(* Logix 5000 project; controller RSL5k_18_Template_noLib Emulate 5570 rev 32.11; software revision 32.02; part 14 of 16 *)
(* tags used below, declared in another part *)
   Inp_SpeedFdbk : REAL;   // Speed Feedbak in Drive Units (typ. 0-32767 = 0 to max freq.)
   Inp_Ready : BOOL;   // 1=Drive is ready to run
   Inp_Running : BOOL;   // 1=Drive is Running (active)
   Inp_CommandDir : BOOL;   // 1=Drive is commanded Forward, 0=Drive is commanded Reverse
   Inp_ActualDir : BOOL;   // 1=Drive is running Forward, 0=Drive is running Reverse
   Inp_FwdPermOK : BOOL;   // 1=Permissives OK, drive can start Forward
   Inp_FwdNBPermOK : BOOL;   // 1=Non-Bypassable Permissives OK, drive can start Forward
   Inp_RevPermOK : BOOL;   // 1=Permissives OK, drive can start Reverse
   Inp_RevNBPermOK : BOOL;   // 1=Non-Bypassable Permissives OK, motor can start Reverse
   Inp_IntlkOK : BOOL;   // 1=Interlocks OK, drive can start/run
   Inp_NBIntlkOK : BOOL;   // 1=Non-Bypassable Interlocks OK, drive can start/run
   Inp_IOFault : BOOL;   // Input Communication Status 0=OK, 1=fail
   Inp_Sim : BOOL;   // 1=Simulate working drive; 0=Start/Stop/ Monitor actual drive
   Inp_OvrdCmd : DINT;   // Override Command: 0=None, 1=Stop, 2=Start Fwd 3=Start Rev
   Cfg_HasRunFdbk : BOOL;   // 1=Drive provides feedback signal on Inp_Running when running
   Cfg_HasSpeedFdbk : BOOL;   // 1=Drive provides speed feedback on Inp_SpeedFdbk
   Cfg_UseSpeedFdbk : BOOL;   // 1=Drive speed determines running state, 0=state determined by drive Active input bit
   Cfg_HasFwdPermObj : BOOL;   // 1=Tells HMI a P_Perm is connected to Inp_FwdPerm
   Cfg_HasRevPermObj : BOOL;   // 1=Tells HMI a P_Perm is connected to Inp_RevPerm
   Cfg_HasIntlkObj : BOOL;   // 1=Tells HMI a P_Intlk is connected to Inp_Intlk
   Cfg_HasResInhObj : BOOL;   // 1=Tells HMI a P_ResInh Restart Inhibit is connected
   Cfg_HasRunTimeObj : BOOL;   // 1=Tells HMI a P_RunTime is connected
   Cfg_SetTrack : BOOL;   // 1=Settings track for unselected sources, 0=no tracking
   Cfg_ShedOnFailToStart : BOOL;   // 1=Stop Motor and Alarm on Fail to Start; 0=Alarm only on Fail to Start
   Cfg_ShedOnIOFault : BOOL;   // 1=Stop Motor and Alarm on I/O Fault; 0=Alarm only on I/O Fault
   Cfg_DecPlcs : DINT;   // Number of decimal places for speed ref/fdbk display (0..6)
   Cfg_InpDLDecPlcs : DINT;   // Number of decimal places for Input Datalink display (0..6)
   Cfg_OutDLDecPlcs : DINT;   // Number of decimal places for Output Datalink display (0..6)
   Cfg_HasDriveFaultAlm : ALIAS FOR DriveFault.Cfg_Exists;   // 1=Drive Fault alarm exists and will be checked
   Cfg_DriveFaultResetReqd : ALIAS FOR DriveFault.Cfg_ResetReqd;   // 1=Reset required to clear Drive Fault Alarm
   Cfg_FailToStartAckReqd : ALIAS FOR FailToStart.Cfg_AckReqd;   // 1=Acknowledge required for Fail to Start Alarm
   Cfg_FailToStopAckReqd : ALIAS FOR FailToStop.Cfg_AckReqd;   // 1=Acknowledge required for Fail to Stop Alarm
   Cfg_IntlkTripAckReqd : ALIAS FOR IntlkTrip.Cfg_AckReqd;   // 1=Acknowledge required for Interlock Trip Alarm
   Cfg_DriveFaultAckReqd : ALIAS FOR DriveFault.Cfg_AckReqd;   // 1=Acknowledge required for Drive Fault Alarm
   Cfg_IOFaultAckReqd : ALIAS FOR IOFault.Cfg_AckReqd;   // 1=Acknowledge required for I/O Fault Alarm
   Cfg_FailToStartSeverity : ALIAS FOR FailToStart.Cfg_Severity;   // Fail To Start Alarm Severity: 1..250=Low, 251..500=Medium, 501..750=High, 751..1000=Urgent
   Cfg_FailToStopSeverity : ALIAS FOR FailToStop.Cfg_Severity;   // Fail To Stop Alarm Severity: 1..250=Low, 251..500=Medium, 501..750=High, 751..1000=Urgent
   Cfg_IntlkTripSeverity : ALIAS FOR IntlkTrip.Cfg_Severity;   // Interlock Trip Alarm Severity: 1..250=Low, 251..500=Medium, 501..750=High, 751..1000=Urgent
   Cfg_DriveFaultSeverity : ALIAS FOR DriveFault.Cfg_Severity;   // Drive Fault Alarm Severity: 1..250=Low, 251..500=Medium, 501..750=High, 751..1000=Urgent
   Cfg_IOFaultSeverity : ALIAS FOR IOFault.Cfg_Severity;   // I/O Fault Alarm Severity: 1..250=Low, 251..500=Medium, 501..750=High, 751..1000=Urgent
   Cfg_MaxSpdRef : REAL;   // Maximum Speed Reference in EU (for limiting)
   Cfg_SpeedRefRawMax : REAL;   // Speed Reference Maximum in Drive (raw) Units (for scaling)
   Cfg_SpeedRefEUMax : REAL;   // Speed Reference Maximum in Engineering Units (for scaling)
   Cfg_SpeedFdbkRawMax : REAL;   // Speed Feedback Maximum in Drive (raw) Units (for scaling)
   Cfg_SpeedFdbkEUMax : REAL;   // Speed Feedback Maximum in Engineering Units (for scaling)
   Cfg_InpDatalinkRawMax : REAL;   // Input Datalink Maximum in Drive (raw) Units (for scaling)
   Cfg_InpDatalinkEUMax : REAL;   // Input Datalink Maximum in Engineering Units (for scaling)
   Cfg_OutDatalinkMax : REAL;   // Maximum Output Datalink in EU (for limiting)
   Cfg_OutDatalinkRawMax : REAL;   // Output Datalink Maximum in Drive (raw) Units (for scaling)
   Cfg_OutDatalinkEUMax : REAL;   // Output Datalink Maximum in Engineering Units (for scaling)
   Cfg_SimRampT : REAL;   // Time to ramp speed fdbk when in Simulation (sec)
   Cfg_FailToStartT : REAL;   // Time after Start to get Run Feedback before Fault (sec)
   Cfg_FailToStopT : REAL;   // Time after Stop to drop Run Feedback before Fault (sec)
   Cfg_ResetPulseT : REAL;   // Time to pulse Out_Reset to clear drive fault
   Cfg_OperKeep : SINT;   // Oper keeps control in Prog / Ext: .0=Reference, .1=Start/Stop/Fwd/ Rev, .3=OutDatalink
   Cfg_ProgKeep : SINT;   // Prog keeps control in Oper / Ext: .0=Reference, .1=Start/Stop/Fwd/ Rev, .3=OutDatalink
   Cfg_ExtKeep : SINT;   // Ext keeps control in Prog / Oper: .0=Reference, .1=Start/Stop/Fwd/ Rev, .3=OutDatalink
   PSet_SpeedRef : REAL;   // Program Setting of Speed Reference (EU)
   PSet_Owner : DINT;   // Program Owner Request ID (non-zero) or Release (zero)
   XSet_SpeedRef : REAL;   // External Setting of Speed Reference (EU)
   PCmd_StartFwd : BOOL;   // Program Command to Start Drive Forward
   PCmd_StartRev : BOOL;   // Program Command to Start Drive Reverse
   PCmd_Stop : BOOL;   // Program Command to Stop Drive
   PCmd_Reset : BOOL;   // Program Command to Reset drive fault and all Alarms requiring Reset
   XCmd_StartFwd : BOOL;   // External Command to Start Drive Forward
   XCmd_StartRev : BOOL;   // External Command to Start Drive Reverse
   XCmd_Stop : BOOL;   // External Command to Stop Drive
   XCmd_JogFwd : BOOL;   // External Command to Jog Drive Forward
   XCmd_JogRev : BOOL;   // External Command to Jog Drive Reverse
   XCmd_Reset : BOOL;   // Ext Cmd to clear shed latches and cleared alarms
   Out_SpeedRef : REAL;   // Drive Speed Reference in Drive Units (typ. 0-32767 = 0 to max freq.)
   Out_Datalink : REAL;   // Auxiliary Signal (datalink) Output in Drive (raw) Units
   Out_Run : BOOL;   // 1=Start/Run Drive, 0=Stop Drive (for held starter type)
   Out_Stop : BOOL;   // 1=Stop Drive, 0=drive left in current state
   Out_Start : BOOL;   // 1=Start Drive, 0=drive left in current state
   Out_Jog : BOOL;   // 1=Jog drive at Jog Speed, -->0=stop jogging
   Out_ClearFault : BOOL;   // 1=Attempt to clear Drive Fault
   Out_Fwd : BOOL;   // 1=Set drive direction to Forward
   Out_Rev : BOOL;   // 1=Set drive direction to Reverse
   Out_Horn : BOOL;   // 1=Sound audible prior to commanded motor start
   Val_SpeedRef : REAL;   // Speed Reference (target) to drive
   Val_SpeedFdbk : REAL;   // Speed Feedback (actual) from drive
   Val_SpeedRefEUMax : REAL;   // Maximum of Speed Reference = MAX (Cfg_SpeedFdbkEUMin, Cfg_SpeedFdbkEUMax)
   Val_SpeedFdbkEUMax : REAL;   // Maximum of Speed Feedback = MAX (Cfg_SpeedFdbkEUMin, Cfg_SpeedFdbkEUMax)
   SrcQ_IO : DINT;   // Source and Quality of primary I/O (enumeration)
   SrcQ : DINT;   // Source and Quality of primary Val/Sts (enumeration)
   Val_Cmd : DINT;   // Device Command 0=None, 1=Stop, 2=StartFwd 3=StartRev 4=JogFwd 5=JogRev
   Val_Fdbk : DINT;   // Device Feedback 0=Stopped, 1=Running Fwd 2=Running Rev 3=Accelerating 4=Decelerating
   Val_Sts : DINT;   // Device Sts: 0=? 1=Stopped 2=RunFwd 3=RunRev 4=RunSlow 5=StartFwd 6=StartRev 7=StartSlow 8=JogFwd 9=JogRev 10=Stopping
   Val_Fault : DINT;   // Device Fault Status 0=None, 16=Fail to Start, 17 = Fail to Stop, 18=Drive Fault, 32=I/O Fault, 34=Config Error
   Val_NotifyAll : DINT;   // Highest Alarm prio and ack status this object + channel (enum)
   Val_UnackAlmC : DINT;   // Count of Unacknowledged Alarms
   Val_Owner : DINT;   // Current Object Owner ID (0=not owned)
   Sts_Stopped : BOOL;   // 1=Drive requested to stop and is confirmed stopped
   Sts_StartingFwd : BOOL;   // 1=Drive requested to run forward and awaiting run feedback
   Sts_StartingRev : BOOL;   // 1=Drive requested to run reverse and awaiting run feedback
   Sts_RunningFwd : BOOL;   // 1=Drive requested to run and is confirmed running forward
   Sts_RunningRev : BOOL;   // 1=Drive requested to run and is confirmed running reverse
   Sts_StoppingFwd : BOOL;   // 1=Drive running forward requested to stop and awaiting stopped feedback
   Sts_StoppingRev : BOOL;   // 1=Drive running reverse requested to stop and awaiting stopped feedback
   Sts_JoggingFwd : BOOL;   // 1=Drive requested to Jog Forward
   Sts_JoggingRev : BOOL;   // 1=Drive requested to Jog Reverse
   Sts_Horn : BOOL;   // 1=Motor Horn Active
   Sts_CommandDir : BOOL;   // 1=Drive commanded to Forward, 0=Reverse
   Sts_ActualDir : BOOL;   // 1=Drive Actual direction is Forward, 0=Reverse
   Sts_Available : BOOL;   // 1=Drive available for control by automation (Prog)
   Nrdy_CfgErr : BOOL;   // 1=Device Not Ready: Configuration Error
   Nrdy_Fail : BOOL;   // 1=Device Not Ready: Device Failure (Shed Requires Reset)
   Nrdy_IOFault : BOOL;   // 1=Device Not Ready: I/O Fault (Shed Requires Reset)
   Nrdy_PrioStop : BOOL;   // 1=Device Not Ready: Oper/Ext Priority Stop Requires Reset
   Nrdy_Trip : BOOL;   // 1=Device not Ready: Deivce Tripped (Drive Fault)
   Sts_Err : BOOL;   // 1=Error in Config: see detail bits for reason
   Err_Alarm : BOOL;   // 1=Error in Config: Alarm Min On Time, Shelf Time, Severity
   Err_FdbkRaw : BOOL;   // 1=Erron in Config: Speed Fdbk Raw Min = Max
   Err_FdbkEU : BOOL;   // 1=Error in Config: Speed Fdbk EU Min = Max
   Sts_Prog : ALIAS FOR CmdSrc.Sts_Prog;
   Sts_Oper : ALIAS FOR CmdSrc.Sts_Oper;
   Sts_Normal : ALIAS FOR CmdSrc.Sts_Normal;
   Sts_ExtReqInh : ALIAS FOR CmdSrc.Sts_ExtReqInh;
   Sts_RdyReset : ALIAS FOR ORdy_Reset;   // 1=A latched alarm or shed condition is ready to be reset
   Sts_RdyAck : BOOL;   // 1=An alarm is ready to be acknowledged
   Ack_FailToStart : ALIAS FOR FailToStart.Ack;   // 1=Fail to Start Alarm has been acknowledged
   Sts_FailToStop : ALIAS FOR FailToStop.Inp;   // 1=Drive Failed to Stop
   Ack_FailToStop : ALIAS FOR FailToStop.Ack;   // 1=Fail to Stop Alarm has been acknowledged
   Ack_IntlkTrip : ALIAS FOR IntlkTrip.Ack;   // 1=Interlock Trip Alarm has been acknowledged
   Sts_DriveFault : ALIAS FOR DriveFault.Inp;   // 1=Drive Fault (see drive display or manual)
   Ack_DriveFault : ALIAS FOR DriveFault.Ack;   // 1=Drive Fault Alarm has been acknowledged
   Sts_IOFault : ALIAS FOR IOFault.Inp;   // I/O Comm Fault Status (0=OK, 1=Bad)
   Ack_IOFault : ALIAS FOR IOFault.Ack;   // 1=I/O Fault Alarm has been acknowledged
   P_VSD : BOOL;   // Unique Parameter Name for auto - discovery
   IOFault : P_Alarm;   // I/O Fault Alarm
   IntlkTrip : P_Alarm;   // Interlock Trip Alarm
   FailToStop : P_Alarm;   // Drive Failed to Stop Alarm
   FailToStart : P_Alarm;   // Drive Failed to Start Alarm
   Wrk_Run : BOOL;   // 1=Drive should be "running", 0=should be "stopped"
   Wrk_Notify : DINT;   // Buffer for building Val_Notify
   DriveFault : P_Alarm;   // Drive Faulted Alarm
   Wrk_Jog : BOOL;   // 1=Jog Drive, 0=Drive not jogging
   Wrk_Sts : DINT;   // Buffer for building Val_Sts
   Wrk_Fault : DINT;   // Buffer for building Val_Fault
   Wrk_SrcQ : DINT;   // Register for building Source / Quality enumeration
   Val_Notify : DINT;   // Current Alarm Level and Acknowledgement (enumeration)
   Wrk_UnackAlmC : DINT;   // Buffer for building Val_UnackAlmC
   OCmd_ResetAckAll : BOOL;   // Oper Cmd to reset shed latches and cleared alarms, plus Acknowledge alarms
   OCmd_Reset : BOOL;   // Oper Cmd to clear shed latches and cleared alarms
   OCmd_JogRev : BOOL;   // Operator Command to Jog Drive Reverse (not cleared by instruction!)
   OCmd_JogFwd : BOOL;   // Operator Command to Jog Drive Forward (not cleared by instruction!)
   OCmd_Stop : BOOL;   // Operator Command to Stop Drive
   OCmd_StartRev : BOOL;   // Operator Command to Start Drive Reverse
   OCmd_StartFwd : BOOL;   // Operator Command to Start Drive Forward
   MCmd_Check : BOOL;   // Maintenance Command to Check (not bypass) all Interlocks and Permissives
   MCmd_Bypass : BOOL;   // Maintenance Command to Bypass all Bypassable Interlocks and Permissives
   ORdy_ResetAckAll : BOOL;   // 1=Ready for OCmd_ResetAckAll (enables HMI button)
   ORdy_Reset : BOOL;   // 1=Ready for OCmd_Reset (enables HMI button)
   ORdy_JogRev : BOOL;   // 1=Ready for OCmd_JogRev (enabled HMI button)
   ORdy_JogFwd : BOOL;   // 1=Ready for OCmd_JogFwd (enables HMI button)
   ORdy_Stop : BOOL;   // 1=Ready for OCmd_Stop (enables HMI button)
   ORdy_StartRev : BOOL;   // 1=Ready for OCmd_StartRev (enables HMI button)
   ORdy_StartFwd : BOOL;   // 1=Ready for OCmd_StartFwd (enables HMI button)
   ORdy_SpeedRef : BOOL;   // 1=Ready for OSet_SpeedRef (enables data entry field)
   MRdy_Check : BOOL;   // 1=Ready for MCmd_Check (enables HMI button)
   MRdy_Bypass : BOOL;   // 1=Ready for MCmd_Bypass (enables HMI button)
(* P_VSD, continued *)

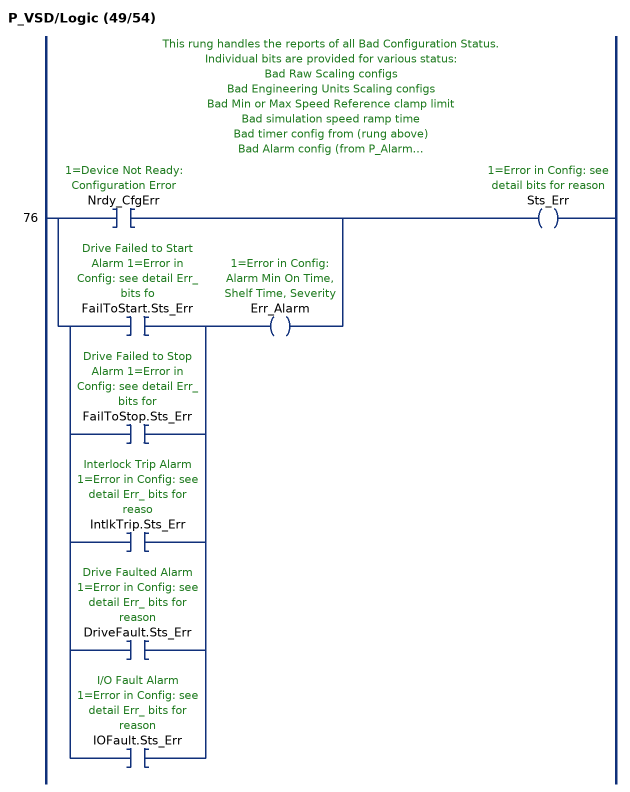
   // This rung handles the reports of all Bad Configuration Status.
   // Individual bits are provided for various status:
   // Bad Raw Scaling configs
   // Bad Engineering Units Scaling configs
   // Bad Min or Max Speed Reference clamp limit
   // Bad simulation speed ramp time
   // Bad timer config from (rung above)
   // Bad Alarm config (from P_Alarm)
   // Bad Cfg_OperKeep / Cfg_ProgKeep config
   // Then a summary Bad Config status is provided, simply an OR of the individual bits.
   // #####  V4.00.00  2018-07-13:  Modified to allow the special case where min and max clamping  #####
   // #####  limits (speed or output datalink) can be EQUAL (clamp at a specific value).  #####
   // #####  Changed delay / time configuration items to REAL seconds.  #####
   76: [XIC(Nrdy_CfgErr) ,[XIC(FailToStart.Sts_Err) ,XIC(FailToStop.Sts_Err) ,XIC(IntlkTrip.Sts_Err) ,XIC(DriveFault.Sts_Err) ,XIC(IOFault.Sts_Err) ] OTE(Err_Alarm) ]OTE(Sts_Err);
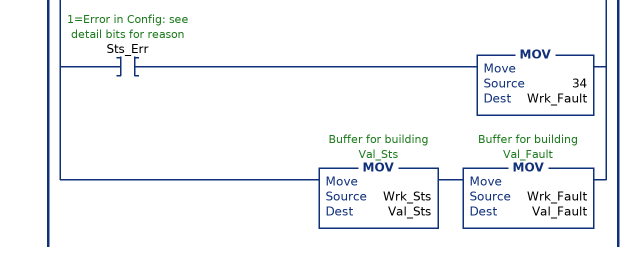
   // Val_Sts is the current device status, as determined by this AOI,
   // based on its knowledge of commands executed and feedback.
   // (This is the status that should be monitored by, for example, FT Historian.)
   // 0 = Powerup / Unknown (in Hand but having no feedback, for example)
   // 0 = Powerup / Unknown
   // 1 = Stopped
   // 2 = Running Forward
   // 3 = Running Reverse
   // 4 = Running Slow
   // 5 = Starting Forward
   // 6 = Starting Reverse
   // 7 = Starting Slow
   // 8 = Jogging Forward
   // 9 = Jogging Reverse
   // 10 = Stopping
   // 14 = Horn
   // Val_Fault is the current device fault status, as determined by this AOI,
   // based on its knowledge of commands executed and feedback.
   // (This is the fault status that should be monitored by, for example, FT Historian.)
   // 0 = None
   // 16 = Fail to Start
   // 17 = Fail to Stop
   // 18 = Drive Fault
   // 32 = I/O Fault (from Input)
   // 34 = Configuration Error
   // #####  V4.00.00 2018-07-13:  Changed Start / Stop / Jog / Fwd / Rev to StartFwd / StartRev / Stop / JogFwd / JogRev  #####
   // #####  Disable/Enable replaced by P_CmdSrc Out of Service (OoS).  #####
   // #####  V4.10.00  2019-03-25:  Added Horn Status.  #####
   77: [CLR(Wrk_Sts) CLR(Wrk_Fault) ,XIC(Sts_Stopped) MOV(1,Wrk_Sts) ,XIC(Sts_RunningFwd) MOV(2,Wrk_Sts) ,XIC(Sts_RunningRev) MOV(3,Wrk_Sts) ,XIC(Sts_StartingFwd) MOV(5,Wrk_Sts) ,XIC(Sts_StartingRev) MOV(6,Wrk_Sts) ,XIC(Sts_JoggingFwd) MOV(8,Wrk_Sts) ,XIC(Sts_JoggingRev) MOV(9,Wrk_Sts) ,[XIC(Sts_StoppingFwd) ,XIC(Sts_StoppingRev) ] MOV(10,Wrk_Sts) ,XIC(Sts_Horn) MOV(14,Wrk_Sts) ,XIC(Nrdy_Fail) MOV(16,Wrk_Fault) ,XIC(Sts_FailToStop) MOV(17,Wrk_Fault) ,XIC(Sts_DriveFault) MOV(18,Wrk_Fault) ,[XIC(Sts_IOFault) ,XIC(Nrdy_IOFault) ] MOV(32,Wrk_Fault) ,XIC(Sts_Err) MOV(34,Wrk_Fault) ,MOV(Wrk_Sts,Val_Sts) MOV(Wrk_Fault,Val_Fault) ];
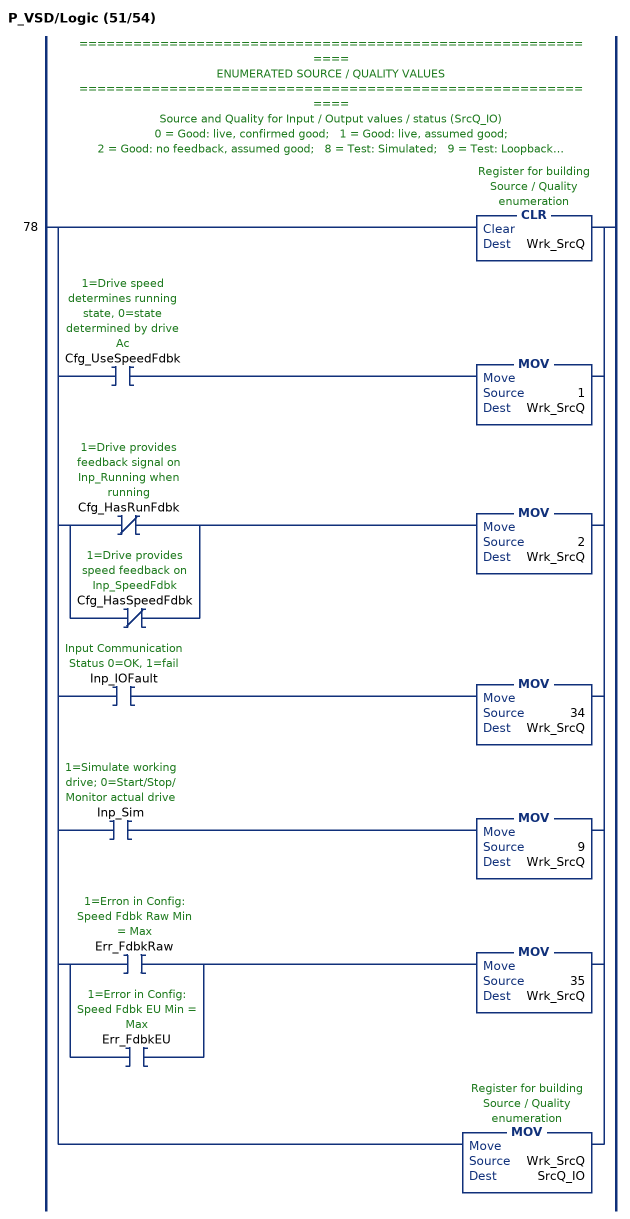
   // ============================================================
   // ENUMERATED SOURCE / QUALITY VALUES
   // ============================================================
   // Source and Quality for Input / Output values / status (SrcQ_IO)
   // 0 = Good: live, confirmed good;   1 = Good: live, assumed good;
   // 2 = Good: no feedback, assumed good;   8 = Test: Simulated;   9 = Test: Loopback;
   // 10 = Test: Manually Entered;   16 = Uncertain: Live, off-spec;
   // 17 = Uncertain, Substituted at Device / Bus;   18 = Uncertain, Substituted at AOI;
   // 19 = Uncertain, using last known good;    20 = Uncertain, using replacement value;
   // 32 = Bad, Signal Failure;   33 = Bad, Channel Fault;
   // 34 = Bad, Module / Comms Fault;   35 = Bad, Invalid Configuration
   78: [CLR(Wrk_SrcQ) ,XIC(Cfg_UseSpeedFdbk) MOV(1,Wrk_SrcQ) ,[XIO(Cfg_HasRunFdbk) ,XIO(Cfg_HasSpeedFdbk) ] MOV(2,Wrk_SrcQ) ,XIC(Inp_IOFault) MOV(34,Wrk_SrcQ) ,XIC(Inp_Sim) MOV(9,Wrk_SrcQ) ,[XIC(Err_FdbkRaw) ,XIC(Err_FdbkEU) ] MOV(35,Wrk_SrcQ) ,MOV(Wrk_SrcQ,SrcQ_IO) ];
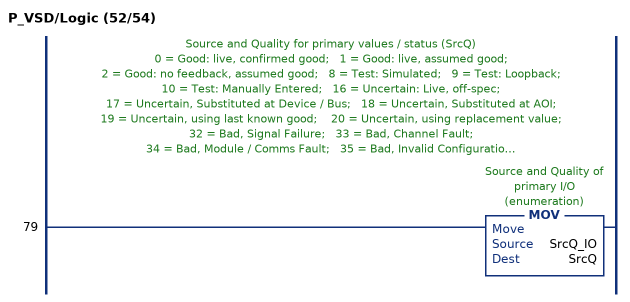
   // Source and Quality for primary values / status (SrcQ)
   // 0 = Good: live, confirmed good;   1 = Good: live, assumed good;
   // 2 = Good: no feedback, assumed good;   8 = Test: Simulated;   9 = Test: Loopback;
   // 10 = Test: Manually Entered;   16 = Uncertain: Live, off-spec;
   // 17 = Uncertain, Substituted at Device / Bus;   18 = Uncertain, Substituted at AOI;
   // 19 = Uncertain, using last known good;    20 = Uncertain, using replacement value;
   // 32 = Bad, Signal Failure;   33 = Bad, Channel Fault;
   // 34 = Bad, Module / Comms Fault;   35 = Bad, Invalid Configuration
   // If the drive is using run feedback (for state) and has speed feedback, all is live and good.
   // If the drive is using speed feedback to determine run state, state is assumed good.
   // If the drive does not have speed feedback, speed is no-feedback assumed good.
   79: MOV(SrcQ_IO,SrcQ);
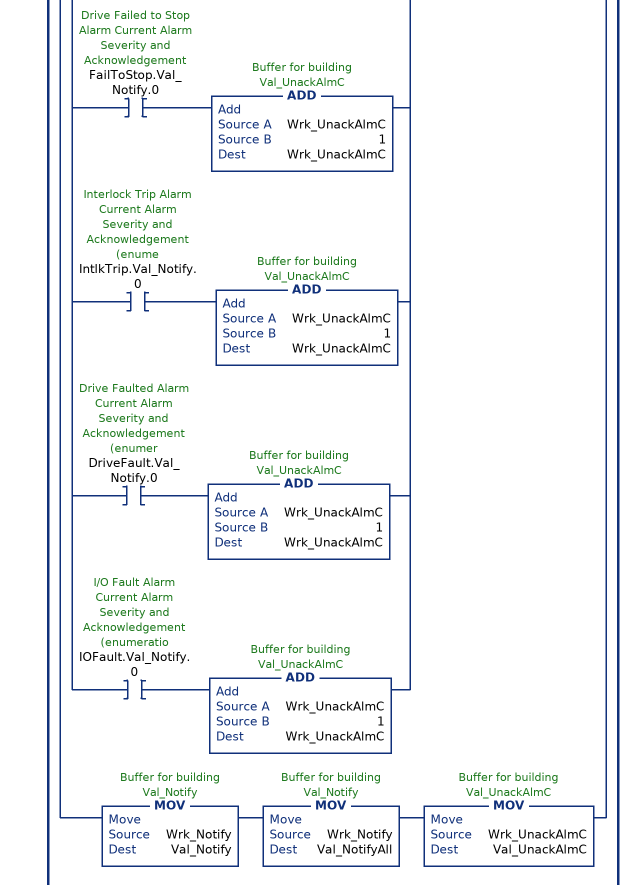
   // ============================================================
   // NOTIFICATION VALUE
   // ============================================================
   // Indicate the current alarm notification level as the max of any of the alarms,
   // and set the low-order bit for reset or ack required:
   // 0 = Not in alarm, acknowledged
   // 1 = Not in alarm, unacknowledged or reset required
   // 2 = Low severity alarm, acknowledged
   // 3 = Low severity alarm, unacknowledged
   // 4 = Medium severity alarm, acknowledged
   // 5 = Medium severity alarm, unacknowledged
   // 6 = High severity alarm, acknowledged
   // 7 = High severity alarm, unacknowledged
   // 8 = Urgent severity alarm, acknowledged
   // 9 = Urgent severity alarm, unacknowledged
   // #####  V4.00.00  2018-07-13:  Added Val_NotifyAll and Val_UnackAlmC to roll up alarm  #####
   // #####  priority / ack status and unack. alarm count.  #####
   80: [CLR(Wrk_Notify) CLR(Wrk_UnackAlmC) ,GRT(FailToStart.Val_Notify,Wrk_Notify) MOV(FailToStart.Val_Notify,Wrk_Notify) ,GRT(FailToStop.Val_Notify,Wrk_Notify) MOV(FailToStop.Val_Notify,Wrk_Notify) ,GRT(IntlkTrip.Val_Notify,Wrk_Notify) MOV(IntlkTrip.Val_Notify,Wrk_Notify) ,GRT(DriveFault.Val_Notify,Wrk_Notify) MOV(DriveFault.Val_Notify,Wrk_Notify) ,GRT(IOFault.Val_Notify,Wrk_Notify) MOV(IOFault.Val_Notify,Wrk_Notify) ,[XIC(FailToStart.Val_Notify.0) ADD(Wrk_UnackAlmC,1,Wrk_UnackAlmC) ,XIC(FailToStop.Val_Notify.0) ADD(Wrk_UnackAlmC,1,Wrk_UnackAlmC) ,XIC(IntlkTrip.Val_Notify.0) ADD(Wrk_UnackAlmC,1,Wrk_UnackAlmC) ,XIC(DriveFault.Val_Notify.0) ADD(Wrk_UnackAlmC,1,Wrk_UnackAlmC) ,XIC(IOFault.Val_Notify.0) ADD(Wrk_UnackAlmC,1,Wrk_UnackAlmC) ] OTE(Wrk_Notify.0) ,MOV(Wrk_Notify,Val_Notify) MOV(Wrk_Notify,Val_NotifyAll) MOV(Wrk_UnackAlmC,Val_UnackAlmC) ];
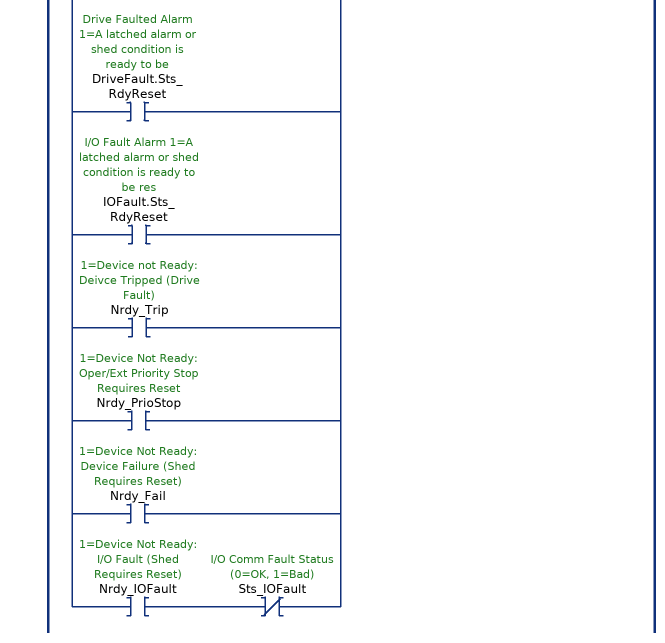
   // This rung identifies:
   // * if a latched Shed condition requires a reset in order to run the motor;
   // * if that reset or any alarm reset or other reset is required; and
   // * if any reset or acknowledge from the operator is required.
   // #####  V4.00.00  2018-07-13:  Aligned ready bit naming with command bit names.  #####
   // #####  All OCmds/MCmds and ORdys/MRdys are now Local Tags.  #####
   // #####  Added Sts_RdyAck and Sts_ResetReqd for use by external objects.  #####
   81: [[XIC(FailToStart.Sts_RdyAck) ,XIC(FailToStop.Sts_RdyAck) ,XIC(IntlkTrip.Sts_RdyAck) ,XIC(IOFault.Sts_RdyAck) ,XIC(DriveFault.Sts_RdyAck) ] OTE(Sts_RdyAck) ,[XIC(FailToStart.Sts_RdyReset) ,XIC(FailToStop.Sts_RdyReset) ,XIC(IntlkTrip.Sts_RdyReset) ,XIC(DriveFault.Sts_RdyReset) ,XIC(IOFault.Sts_RdyReset) ,XIC(Nrdy_Trip) ,XIC(Nrdy_PrioStop) ,XIC(Nrdy_Fail) ,XIC(Nrdy_IOFault) XIO(Sts_IOFault) ] OTE(ORdy_Reset) ]OTE(ORdy_ResetAckAll);
END_ROUTINE

ROUTINE Prescan   (* ladder *)
// Clear Ownership, set drive to STOP, clear "lurking" Commands
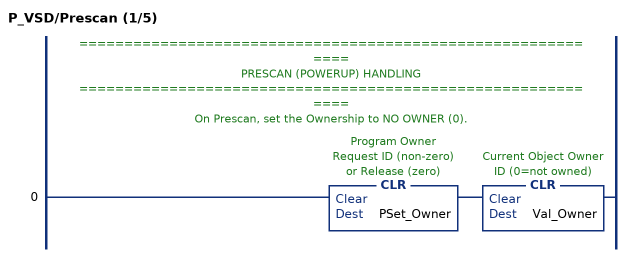
   // ============================================================
   // PRESCAN (POWERUP) HANDLING
   // ============================================================
   // On Prescan, set the Ownership to NO OWNER (0).
   0: CLR(PSet_Owner)CLR(Val_Owner);
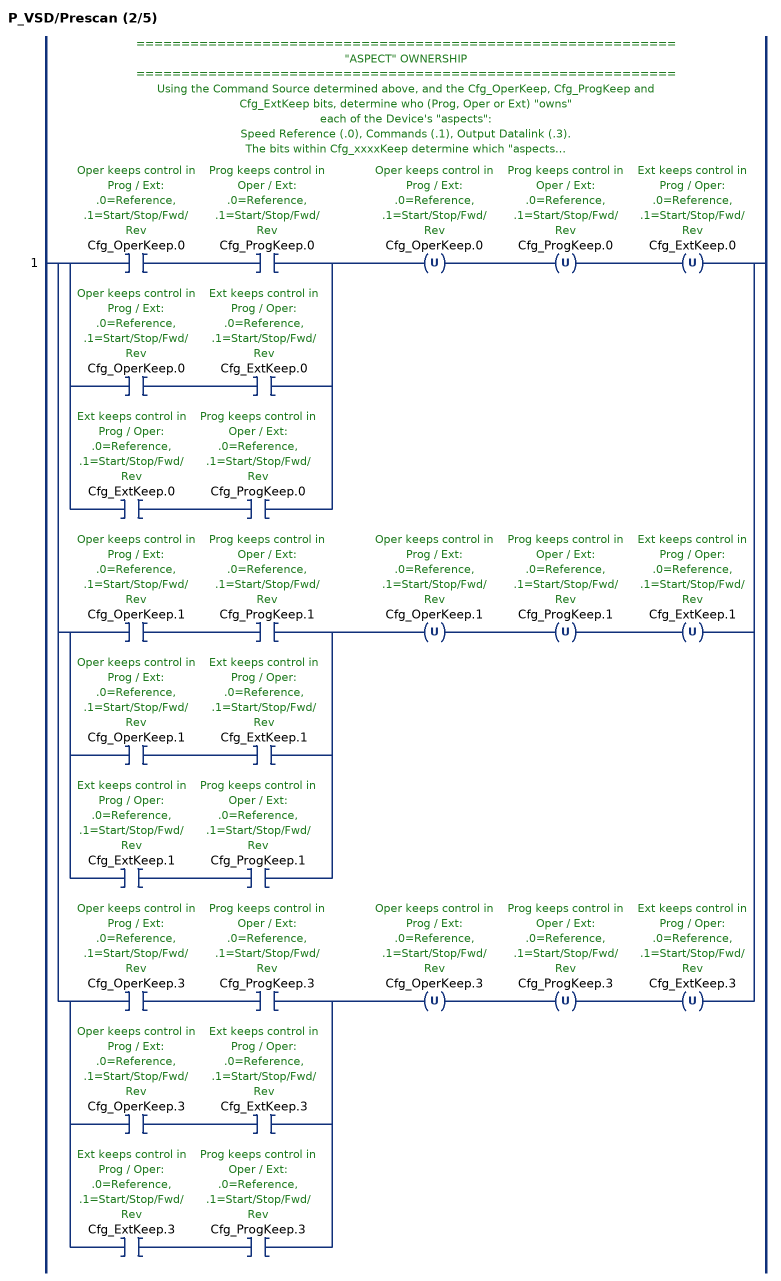
   // ============================================================
   // "ASPECT" OWNERSHIP
   // ============================================================
   // Using the Command Source determined above, and the Cfg_OperKeep, Cfg_ProgKeep and
   // Cfg_ExtKeep bits, determine who (Prog, Oper or Ext) "owns"
   // each of the Device's "aspects":
   // Speed Reference (.0), Commands (.1), Output Datalink (.3).
   // The bits within Cfg_xxxxKeep determine which "aspects"
   // (sub-functions of this AOI) are retained by the Oper, Prog or Ext
   // when one of the other command sources is selected.
   // All aspects (functions) may be "kept" (basically locking the command source
   // slection, rendering it moot --  you get to explain how it works to your operators!!!),
   // but it is NOT allowed to have any given function retained by more than one
   // source.  This rung ensures that no function is "kept" by more than one source.
   // ON PRESCAN:  If any two of Oper Keep, Prog Keep and Ext Keep get set on download or during
   // controller PROG mode, they are ALL CLEARED on powerup!!!
   1: [[XIC(Cfg_OperKeep.0) XIC(Cfg_ProgKeep.0) ,XIC(Cfg_OperKeep.0) XIC(Cfg_ExtKeep.0) ,XIC(Cfg_ExtKeep.0) XIC(Cfg_ProgKeep.0) ] OTU(Cfg_OperKeep.0) OTU(Cfg_ProgKeep.0) OTU(Cfg_ExtKeep.0) ,[XIC(Cfg_OperKeep.1) XIC(Cfg_ProgKeep.1) ,XIC(Cfg_OperKeep.1) XIC(Cfg_ExtKeep.1) ,XIC(Cfg_ExtKeep.1) XIC(Cfg_ProgKeep.1) ] OTU(Cfg_OperKeep.1) OTU(Cfg_ProgKeep.1) OTU(Cfg_ExtKeep.1) ,[XIC(Cfg_OperKeep.3) XIC(Cfg_ProgKeep.3) ,XIC(Cfg_OperKeep.3) XIC(Cfg_ExtKeep.3) ,XIC(Cfg_ExtKeep.3) XIC(Cfg_ProgKeep.3) ] OTU(Cfg_OperKeep.3) OTU(Cfg_ProgKeep.3) OTU(Cfg_ExtKeep.3) ];
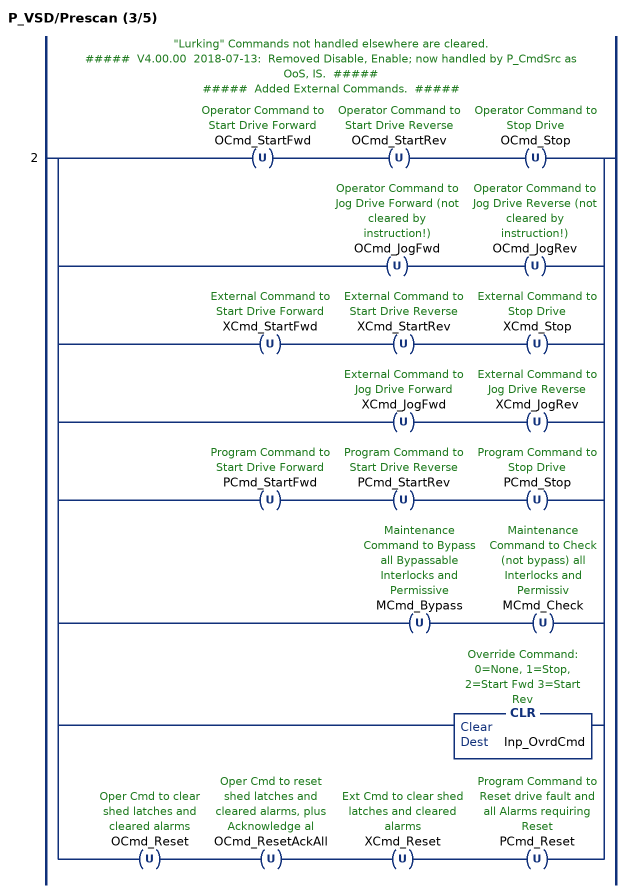
   // "Lurking" Commands not handled elsewhere are cleared.
   // #####  V4.00.00  2018-07-13:  Removed Disable, Enable; now handled by P_CmdSrc as OoS, IS.  #####
   // #####  Added External Commands.  #####
   2: [OTU(OCmd_StartFwd) OTU(OCmd_StartRev) OTU(OCmd_Stop) ,OTU(OCmd_JogFwd) OTU(OCmd_JogRev) ,OTU(XCmd_StartFwd) OTU(XCmd_StartRev) OTU(XCmd_Stop) ,OTU(XCmd_JogFwd) OTU(XCmd_JogRev) ,OTU(PCmd_StartFwd) OTU(PCmd_StartRev) OTU(PCmd_Stop) ,OTU(MCmd_Bypass) OTU(MCmd_Check) ,CLR(Inp_OvrdCmd) ,OTU(OCmd_Reset) OTU(OCmd_ResetAckAll) OTU(XCmd_Reset) OTU(PCmd_Reset) ];
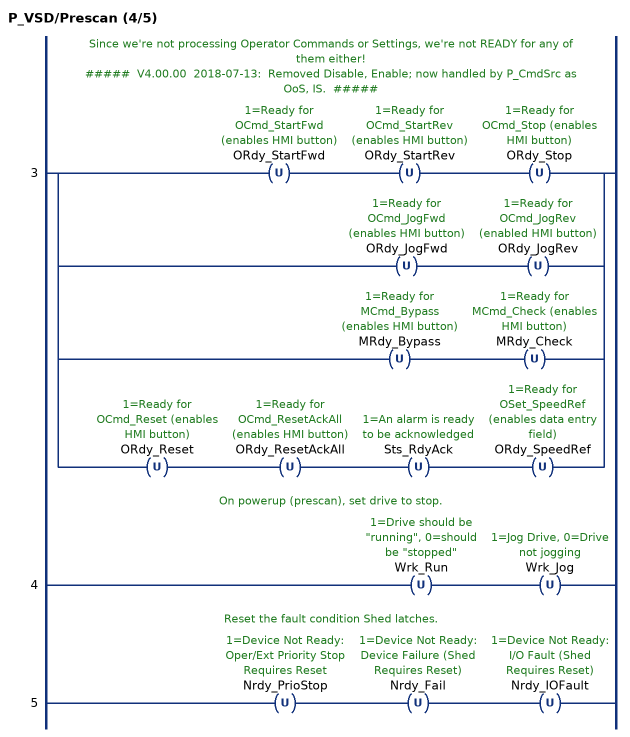
   // Since we're not processing Operator Commands or Settings, we're not READY for any of them either!
   // #####  V4.00.00  2018-07-13:  Removed Disable, Enable; now handled by P_CmdSrc as OoS, IS.  #####
   3: [OTU(ORdy_StartFwd) OTU(ORdy_StartRev) OTU(ORdy_Stop) ,OTU(ORdy_JogFwd) OTU(ORdy_JogRev) ,OTU(MRdy_Bypass) OTU(MRdy_Check) ,OTU(ORdy_Reset) OTU(ORdy_ResetAckAll) OTU(Sts_RdyAck) OTU(ORdy_SpeedRef) ];
   // On powerup (prescan), set drive to stop.
   4: OTU(Wrk_Run)OTU(Wrk_Jog);
   // Reset the fault condition Shed latches.
   5: OTU(Nrdy_PrioStop)OTU(Nrdy_Fail)OTU(Nrdy_IOFault);
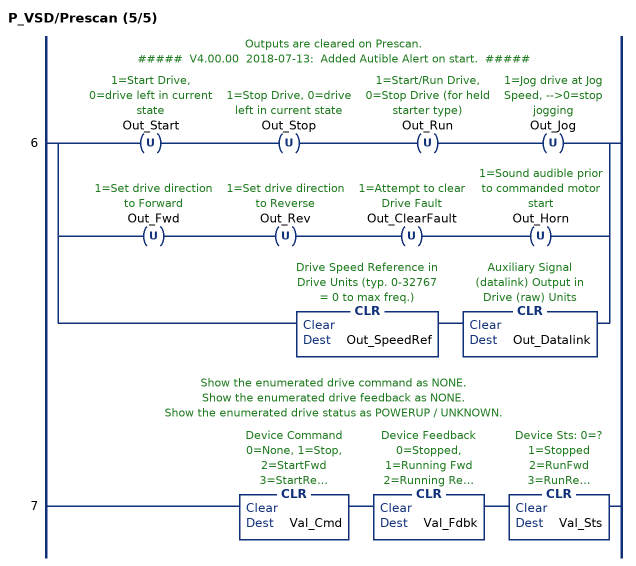
   // Outputs are cleared on Prescan.
   // #####  V4.00.00  2018-07-13:  Added Autible Alert on start.  #####
   6: [OTU(Out_Start) OTU(Out_Stop) OTU(Out_Run) OTU(Out_Jog) ,OTU(Out_Fwd) OTU(Out_Rev) OTU(Out_ClearFault) OTU(Out_Horn) ,CLR(Out_SpeedRef) CLR(Out_Datalink) ];
   // Show the enumerated drive command as NONE.
   // Show the enumerated drive feedback as NONE.
   // Show the enumerated drive status as POWERUP / UNKNOWN.
   7: CLR(Val_Cmd)CLR(Val_Fdbk)CLR(Val_Sts);
END_ROUTINE
END_ADD_ON_INSTRUCTION

VAR_GLOBAL   (* controller tags *)
   E300_TripCodeList : P_DescList[90] := ([0].Desc := 'No Trip Conditions Detected', [1].Code := 1, [1].Desc := 'Motor overcurrent trip', [2].Code := 2, [2].Desc := 'Motor phase loss trip', [3].Code := 3, [3].Desc := 'Ground fault trip', [4].Code := 4, [4].Desc := 'Motor stall (fail to reach speed) trip', [5].Code := 5, [5].Desc := 'Motor current over jam trip limit', [6].Code := 6, [6].Desc := 'Motor current below operating point trip', [7].Code := 7, [7].Desc := 'Phase-to-phase current imbalance trip', [8].Code := 8, [8].Desc := 'L1 undercurrent trip', [9].Code := 9, [9].Desc := 'L2 undercurrent trip', [10].Code := 10, [10].Desc := 'L3 undercurrent trip', [11].Code := 11, [11].Desc := 'L1 overcurrent trip', [12].Code := 12, [12].Desc := 'L2 overcurrent trip', [13].Code := 13, [13].Desc := 'L3 overcurrent trip', [14].Code := 14, [14].Desc := 'L1 current loss trip', [15].Code := 15, [15].Desc := 'L2 current loss trip', [16].Code := 16, [16].Desc := 'L3 current loss trip', [17].Code := 17, [17].Desc := 'Line-to-line undervoltage trip', [18].Code := 18, [18].Desc := 'Line-to line overvoltage trip', [19].Code := 19, [19].Desc := 'Phase-to-phase voltage imbalance trip', [20].Code := 20, [20].Desc := 'Supply voltage phases rotated', [21].Code := 21, [21].Desc := 'Low line frequency trip', [22].Code := 22, [22].Desc := 'High line frequency trip', [23].Code := 25, [23].Desc := 'Sensing module firmware failed to load', [24].Code := 26, [24].Desc := 'Sensing Module output enable open trip', [25].Code := 27, [25].Desc := 'Sensing Module missing interrupts trip', [26].Code := 28, [26].Desc := 'Sensing Module not calibrated trip', [27].Code := 29, [27].Desc := 'Sensing Module frame type failure trip', [28].Code := 30, [28].Desc := 'Sensing Module configuration failure', [29].Code := 31, [29].Desc := 'Sensing Module overrun error trip', [30].Code := 32,
        [30].Desc := 'Sensing Module not responding trip', [31].Code := 33, [31].Desc := 'Low total real power (kW) trip', [32].Code := 34, [32].Desc := 'High total real power (kW) trip', [33].Code := 35, [33].Desc := 'Low reactive pwr consumed (+kVAR) trip', [34].Code := 36, [34].Desc := 'High reactive pwr consumed (+kVAR) trip', [35].Code := 37, [35].Desc := 'Low reactive pwr generated (-kVAR) trip', [36].Code := 38, [36].Desc := 'High reactive pwr generated (-kVAR) trip', [37].Code := 39, [37].Desc := 'Low apparent power (kVA) trip', [38].Code := 40, [38].Desc := 'High apparent power (kVA) trip', [39].Code := 41, [39].Desc := 'Low power factor lagging (-PF) trip', [40].Code := 42, [40].Desc := 'High power factor lagging (-PF) trip', [41].Code := 43, [41].Desc := 'Low power factor leading (+PF) trip', [42].Code := 44, [42].Desc := 'High power factor leading (+PF) trip', [43].Code := 49, [43].Desc := 'Test trip (held Test/Reset button)', [44].Code := 50, [44].Desc := 'Motor stator windings overheated', [45].Code := 51, [45].Desc := 'DeviceLogix defined trip was generated', [46].Code := 52, [46].Desc := 'Stop button pressed at Operator Station', [47].Code := 53, [47].Desc := 'Remote trip commanded', [48].Code := 54, [48].Desc := 'Maximum starts per hour exceeded', [49].Code := 55, [49].Desc := 'Hardware config. fault, check inputs', [50].Code := 58, [50].Desc := 'DeviceLogix feedback timeout trip', [51].Code := 59, [51].Desc := 'Control Module CAN0 init failure', [52].Code := 60, [52].Desc := 'Control Module CAN0 bus failure', [53].Code := 61, [53].Desc := 'Control Module CAN1 init failure', [54].Code := 62, [54].Desc := 'Control Module CAN1 bus failure', [55].Code := 63, [55].Desc := 'Control Module ADC0 failure trip', [56].Code := 64, [56].Desc := 'Control Module CRC error count trip', [57].Code := 65, [57].Desc := 'Analog module 1 channel 00 trip', [58].Code := 66, [58].Desc := 'Analog module 1 channel 01 trip', [59].Code := 67, [59].Desc := 'Analog module 1 channel 02 trip', [60].Code := 68,
        [60].Desc := 'Analog module 2 channel 00 trip', [61].Code := 69, [61].Desc := 'Analog module 2 channel 01 trip', [62].Code := 70, [62].Desc := 'Analog module 2 channel 02 trip', [63].Code := 71, [63].Desc := 'Analog module 3 channel 00 trip', [64].Code := 72, [64].Desc := 'Analog module 3 channel 01 trip', [65].Code := 73, [65].Desc := 'Analog module 3 channel 02 trip', [66].Code := 74, [66].Desc := 'Analog module 4 channel 00 trip', [67].Code := 75, [67].Desc := 'Analog module 4 channel 01 trip', [68].Code := 76, [68].Desc := 'Analog module 4 channel 02 trip', [69].Code := 77, [69].Desc := 'Ext. NVS Chip comms timeout trip', [70].Code := 78, [70].Desc := 'Ext. NVS CRC error trip', [71].Code := 79, [71].Desc := 'Ext. NVS Chip data out of range trip', [72].Code := 81, [72].Desc := 'Digital exp. module 1 malfunction trip', [73].Code := 82, [73].Desc := 'Digital exp. module 2 malfunction trip', [74].Code := 83, [74].Desc := 'Digital exp. module 3 malfunction trip', [75].Code := 84, [75].Desc := 'Digital exp. module 4 malfunction trip', [76].Code := 85, [76].Desc := 'Analog exp. module 1 malfunction trip', [77].Code := 86, [77].Desc := 'Analog exp. module 2 malfunction trip', [78].Code := 87, [78].Desc := 'Analog exp. module 3 malfunction trip', [79].Code := 88, [79].Desc := 'Analog exp. module 4 malfunction trip', [80].Code := 90, [80].Desc := 'Control module type mismatch trip', [81].Code := 91, [81].Desc := 'Sensing module type mismatch trip', [82].Code := 92, [82].Desc := 'Communication module type mismatch trip', [83].Code := 93, [83].Desc := 'Operator station type mismatch trip', [84].Code := 94, [84].Desc := 'Digital I/O module type mismatch trip', [85].Code := 95, [85].Desc := 'Analog I/O module type mismatch trip', [86].Code := 96, [86].Desc := 'Current/voltage detected in Test Mode', [87].Code := 97, [87].Desc := 'Heap memory could not be allocated', [88].Code := 98, [88].Desc := 'Vendor ID hardware fault');   // E300 Overload Relay Trip History Codes and Descriptions
   E300_WarningCodeList : P_DescList[67] := ([0].Desc := 'No warnings', [1].Code := 1, [1].Desc := 'Approaching motor current overload', [2].Code := 3, [2].Desc := 'Motor lead or winding ground fault', [3].Code := 5, [3].Desc := 'Motor current over jam warning limit', [4].Code := 6, [4].Desc := 'Motor below normal operating current', [5].Code := 7, [5].Desc := 'Phase-t0-phase current imbalance warning', [6].Code := 8, [6].Desc := 'L1 undercurrent warning', [7].Code := 9, [7].Desc := 'L2 undercurrent warning', [8].Code := 10, [8].Desc := 'L3 undercurrent warning', [9].Code := 11, [9].Desc := 'L1 overcurrent warning', [10].Code := 12, [10].Desc := 'L2 overcurrent warning', [11].Code := 13, [11].Desc := 'L3 overcurrent warning', [12].Code := 14, [12].Desc := 'L1 current loss warning', [13].Code := 15, [13].Desc := 'L2 current loss warning', [14].Code := 16, [14].Desc := 'L3 current loss warning', [15].Code := 17, [15].Desc := 'Line-to-line undervoltage warning', [16].Code := 18, [16].Desc := 'Line-to-line overvoltage warning', [17].Code := 19, [17].Desc := 'Phase-to-phase voltage imbalance warning', [18].Code := 20, [18].Desc := 'Supply voltage phases rotated warning', [19].Code := 21, [19].Desc := 'Low line frequency warning', [20].Code := 22, [20].Desc := 'High line frequency warning', [21].Code := 33, [21].Desc := 'Low total real power (kW) warning', [22].Code := 34, [22].Desc := 'High total real power (kW) warning', [23].Code := 35, [23].Desc := 'Low reactive pwr consumed (+kVAR) warn', [24].Code := 36, [24].Desc := 'High reactive pwr consumed (+kVAR) warn', [25].Code := 37, [25].Desc := 'Low reactive pwr generated (-kVAR) warn', [26].Code := 38, [26].Desc := 'High reactive pwr generated (-kVAR) warn', [27].Code := 39, [27].Desc := 'Low apparent power (kVA) warning', [28].Code := 40, [28].Desc := 'High apparent power (kVA) warning', [29].Code := 41, [29].Desc := 'Low power factor lagging (-PF) warning', [30].Code := 42,
        [30].Desc := 'High power factor lagging (-PF) warning', [31].Code := 43, [31].Desc := 'Low power factor leading (+PF) warning', [32].Code := 44, [32].Desc := 'High power factor leading (+PF) warning', [33].Code := 50, [33].Desc := 'Motor stator windings overheated (PTC)', [34].Code := 51, [34].Desc := 'DeviceLogix defined warning', [35].Code := 56, [35].Desc := 'Config Error, see par. 38-39 for reason', [36].Code := 58, [36].Desc := 'DeviceLogix feedback timeout trip', [37].Code := 60, [37].Desc := 'Number of starts warning', [38].Code := 61, [38].Desc := 'Operating hours warning', [39].Code := 65, [39].Desc := 'Analog module 1 channel 00 warning', [40].Code := 66, [40].Desc := 'Analog module 1 channel 01 warning', [41].Code := 67, [41].Desc := 'Analog module 1 channel 02 warning', [42].Code := 68, [42].Desc := 'Analog module 2 channel 00 warning', [43].Code := 69, [43].Desc := 'Analog module 2 channel 01 warning', [44].Code := 70, [44].Desc := 'Analog module 2 channel 02 warning', [45].Code := 71, [45].Desc := 'Analog module 3 channel 00 warning', [46].Code := 72, [46].Desc := 'Analog module 3 channel 01 warning', [47].Code := 73, [47].Desc := 'Analog module 3 channel 02 warning', [48].Code := 74, [48].Desc := 'Analog module 4 channel 00 warning', [49].Code := 75, [49].Desc := 'Analog module 4 channel 01 warning', [50].Code := 76, [50].Desc := 'Analog module 4 channel 02 warning', [51].Code := 81, [51].Desc := 'Digital expansion module 1 malfunction', [52].Code := 82, [52].Desc := 'Digital expansion module 2 malfunction', [53].Code := 83, [53].Desc := 'Digital expansion module 3 malfunction', [54].Code := 84, [54].Desc := 'Digital expansion module 4 malfunction', [55].Code := 85, [55].Desc := 'Analog expansion module 1 malfunction', [56].Code := 86, [56].Desc := 'Analog expansion module 2 malfunction', [57].Code := 87, [57].Desc := 'Analog expansion module 3 malfunction', [58].Code := 88, [58].Desc := 'Analog expansion module 4 malfunction', [59].Code := 90, [59].Desc := 'Control module type mismatch', [60].Code := 91,
        [60].Desc := 'Sensing module type mismatch', [61].Code := 92, [61].Desc := 'Communication module type mismatch', [62].Code := 93, [62].Desc := 'Operator station type mismatch', [63].Code := 94, [63].Desc := 'Digital I/O module type mismatch', [64].Code := 95, [64].Desc := 'Analog I/O module type mismatch', [65].Code := 98, [65].Desc := 'Hardware fault');   // E300 Overload Relay Warning History Codes and Descriptions
   L_TaskMonitor : L_TaskMon[8] := ([0].Cfg_HasOverPlanAlm := 1, [0].Cfg_OverPlanAckReqd := 1, [0].Cfg_OverPlanSeverity := 3, [0].Cfg_PlanExecT := 3000.0, [0].Sts_TaskInhibited := 1, [0].Ack_OverPlan := 1, [1].Cfg_HasOverPlanAlm := 1, [1].Cfg_OverPlanAckReqd := 1, [1].Cfg_OverPlanSeverity := 3, [1].Cfg_PlanExecT := 3000.0, [1].Val_Rate := 100.00001, [1].Val_Priority := 6, [1].Val_LastExecT := 0.044000003, [1].Val_MaxExecT := 3.9420002, [1].Val_OverlapC := 13, [1].Val_WatchdogT := 300.0, [1].Ack_OverPlan := 1, [2].Cfg_HasOverPlanAlm := 1, [2].Cfg_OverPlanAckReqd := 1, [2].Cfg_OverPlanSeverity := 3, [2].Cfg_PlanExecT := 3000.0, [2].Val_Rate := 250.00002, [2].Val_Priority := 7, [2].Val_LastExecT := 0.066, [2].Val_MaxExecT := 0.98300004, [2].Val_WatchdogT := 750.00006, [2].Ack_OverPlan := 1, [3].Cfg_HasOverPlanAlm := 1, [3].Cfg_OverPlanAckReqd := 1, [3].Cfg_OverPlanSeverity := 3, [3].Cfg_PlanExecT := 3000.0, [3].Val_Rate := 500.00003, [3].Val_Priority := 8, [3].Val_LastExecT := 0.19700001, [3].Val_MaxExecT := 3.7970002, [3].Val_WatchdogT := 1500.0001, [3].Ack_OverPlan := 1, [4].Cfg_HasOverPlanAlm := 1, [4].Cfg_OverPlanAckReqd := 1, [4].Cfg_OverPlanSeverity := 3, [4].Cfg_PlanExecT := 3000.0, [4].Val_Rate := 1000.00006, [4].Val_Priority := 9, [4].Val_LastExecT := 0.031000001, [4].Val_MaxExecT := 0.35700002, [4].Val_WatchdogT := 3000.0002, [4].Ack_OverPlan := 1, [5].Cfg_HasOverPlanAlm := 1, [5].Cfg_OverPlanAckReqd := 1, [5].Cfg_OverPlanSeverity := 3, [5].Cfg_PlanExecT := 3000.0, [5].Val_Rate := 2000.0001, [5].Val_Priority := 10, [5].Val_LastExecT := 0.032, [5].Val_MaxExecT := 0.223, [5].Val_WatchdogT := 6000.0005, [5].Ack_OverPlan := 1, [6].Cfg_HasOverPlanAlm := 1, [6].Cfg_OverPlanAckReqd := 1, [6].Cfg_OverPlanSeverity := 3,
        [6].Cfg_PlanExecT := 3000.0, [6].Val_Rate := 5000.0, [6].Val_Priority := 11, [6].Val_LastExecT := 0.017, [6].Val_MaxExecT := 0.386, [6].Val_WatchdogT := 15000.001, [6].Ack_OverPlan := 1, [7].Cfg_HasOverPlanAlm := 1, [7].Cfg_OverPlanAckReqd := 1, [7].Cfg_OverPlanSeverity := 3, [7].Cfg_PlanExecT := 3000.0, [7].Val_Rate := 10000.0, [7].Val_Priority := 12, [7].Val_LastExecT := 0.017, [7].Val_MaxExecT := 0.18800001, [7].Val_WatchdogT := 30000.002, [7].Ack_OverPlan := 1);
   LC1 : P_PIDE := (Inp_PV := 30.00001, Inp_CVInitVal := 30.00001, Inp_CVPrev := 1.e-45, Inp_IntlkOK := 1, Inp_NBIntlkOK := 1, Inp_OvrdRatio := 1.0, Inp_OvrdSP := 30.0, Inp_OvrdCV := 30.00001, Inp_HiHiDevGate := 1, Inp_HiDevGate := 1, Inp_LoDevGate := 1, Inp_LoLoDevGate := 1, Cfg_HasAuto := 1, Cfg_HasMan := 1, Cfg_PVTrack := 1, Cfg_Depend := 1, Cfg_DerivSPAct := 1, Cfg_SetTrack := 1, Cfg_HasIntlkObj := 1, Cfg_SPFailSPAct := 1, Cfg_IntlkTripCVAct := 2, Cfg_SPFailCVAct := 1, Cfg_PVFailCVAct := 1, Cfg_CVFailCVAct := 1, Cfg_PVDecPlcs := 2, Cfg_CVDecPlcs := 2, Cfg_HiHiDevAckReqd := 1, Cfg_HiDevAckReqd := 1, Cfg_LoDevAckReqd := 1, Cfg_LoLoDevAckReqd := 1, Cfg_IntlkTripAckReqd := 1, Cfg_FailAckReqd := 1, Cfg_HiHiDevSeverity := 501, Cfg_HiDevSeverity := 251, Cfg_LoDevSeverity := 251, Cfg_LoLoDevSeverity := 501, Cfg_IntlkTripSeverity := 251, Cfg_FailSeverity := 751, Cfg_MinRatio := 1.0, Cfg_MaxRatio := 1.0, Cfg_MaxSP := 100.0, Cfg_PVEUMax := 100.0, Cfg_CVEUMax := 100.0, Cfg_CVRawMax := 100.0, Cfg_PGain := 1.135597, Cfg_IGain := 0.16608427, Cfg_MaxCV := 100.0, PSet_Ratio := 1.0, PSet_SP := 30.0, PSet_CV := 30.00001, XSet_Ratio := 1.0, XSet_SP := 30.0, XSet_CV := 30.00001, Out_CV := 30.00001, Val_PV := 30.00001, Val_Ratio := 1.0, Val_SPSet := 30.0, Val_SP := 30.0, Val_E := -9.536743e-06, Val_CVSet := 30.00001,
        Val_CVOut := 30.00001, Val_PVPercent := 30.00001, Val_SPPercent := 30.0, Val_EPercent := -9.536743e-06, Val_CVPercent := 30.00001, Val_ActExecT := 0.501, Val_Init := 30.0, Val_PVEUMax := 100.0, Val_CVEUMax := 100.0, Val_Sts := 2, Val_State := 2, Sts_Auto := 1, Sts_InitReq := 1, Sts_Active := 1, Sts_Oper := 1, Sts_Normal := 1, Sts_ExtReqInh := 1, Sts_HiHiDevGate := 1, Ack_HiHiDev := 1, Sts_HiDevGate := 1, Ack_HiDev := 1, Sts_LoDevGate := 1, Ack_LoDev := 1, Sts_LoLoDevGate := 1, Ack_LoLoDev := 1, Ack_IntlkTrip := 1, Ack_Fail := 1);   // TagDescript
   LC1_Intlk : P_Intlk := (Sts_IntlkOK := 1, Sts_NBIntlkOK := 1);   // TagDescript - Interlocks
   LT1 : P_AIn := (Inp_PV := 30.00001, Inp_HiHiGate := 1, Inp_HiGate := 1, Inp_LoGate := 1, Inp_LoLoGate := 1, Inp_FailGate := 1, Cfg_PVDecPlcs := 2, Cfg_HasLoAlm := 1, Cfg_HiHiAckReqd := 1, Cfg_HiAckReqd := 1, Cfg_LoAckReqd := 1, Cfg_LoLoAckReqd := 1, Cfg_FailAckReqd := 1, Cfg_HiHiSeverity := 501, Cfg_HiSeverity := 251, Cfg_LoSeverity := 251, Cfg_LoLoSeverity := 501, Cfg_FailSeverity := 751, Cfg_InpRawMax := 100.0, Cfg_PVEUMax := 100.0, Cfg_HiHiLim := 1.5e+38, Cfg_HiHiDB := 1.0, Cfg_HiLim := 1.5e+38, Cfg_HiDB := 1.0, Cfg_LoLim := 24.0, Cfg_LoDB := 1.0, Cfg_LoLoLim := -1.5e+38, Cfg_LoLoDB := 1.0, Cfg_FailHiLim := 103.9583, Cfg_FailLoLim := -2.083333, Cfg_FailDB := 0.4166667, Set_SimPV := 30.00001, Val := 30.00001, Val_InpPV := 30.00001, Val_PVMinCapt := 1.4e-44, Val_PVMaxCapt := 30.012833, Val_PVEUMax := 100.0, SrcQ_IO := 1, SrcQ := 1, Val_NotifyAll := 1, Val_UnackAlmC := 1, Sts_RdyAck := 1, Sts_HiHiGate := 1, Ack_HiHi := 1, Sts_HiGate := 1, Ack_Hi := 1, Sts_LoGate := 1, Sts_LoLoGate := 1, Ack_LoLo := 1, Sts_FailGate := 1, Ack_Fail := 1);   // TagDescript
   P1 : P_VSD := (Inp_SpeedFdbk := 7561.6177, Inp_Ready := 1, Inp_CommandDir := 1, Inp_ActualDir := 1, Inp_FwdPermOK := 1, Inp_FwdNBPermOK := 1, Inp_RevPermOK := 1, Inp_RevNBPermOK := 1, Inp_IntlkOK := 1, Inp_NBIntlkOK := 1, Cfg_HasFwdPermObj := 1, Cfg_HasRevPermObj := 1, Cfg_HasIntlkObj := 1, Cfg_HasResInhObj := 1, Cfg_HasRunTimeObj := 1, Cfg_SetTrack := 1, Cfg_ShedOnFailToStart := 1, Cfg_ShedOnIOFault := 1, Cfg_DecPlcs := 2, Cfg_InpDLDecPlcs := 2, Cfg_OutDLDecPlcs := 2, Cfg_HasDriveFaultAlm := 1, Cfg_DriveFaultResetReqd := 1, Cfg_FailToStartAckReqd := 1, Cfg_FailToStopAckReqd := 1, Cfg_IntlkTripAckReqd := 1, Cfg_DriveFaultAckReqd := 1, Cfg_IOFaultAckReqd := 1, Cfg_FailToStartSeverity := 501, Cfg_FailToStopSeverity := 501, Cfg_IntlkTripSeverity := 251, Cfg_DriveFaultSeverity := 751, Cfg_IOFaultSeverity := 751, Cfg_MaxSpdRef := 60.0, Cfg_SpeedRefRawMax := 32767.0, Cfg_SpeedRefEUMax := 130.0, Cfg_SpeedFdbkRawMax := 32767.0, Cfg_SpeedFdbkEUMax := 130.0, Cfg_InpDatalinkRawMax := 4095.0, Cfg_InpDatalinkEUMax := 409.5, Cfg_OutDatalinkMax := 100.0, Cfg_OutDatalinkRawMax := 4095.0, Cfg_OutDatalinkEUMax := 409.5, Cfg_SimRampT := 10.0, Cfg_FailToStartT := 15.0, Cfg_FailToStopT := 15.0, Cfg_ResetPulseT := 2.0, PSet_SpeedRef := 30.00001, XSet_SpeedRef := 30.00001, Out_SpeedRef := 7561.6177, Out_Run := 1, Out_Fwd := 1, Val_SpeedRef := 30.00001, Val_SpeedFdbk := 30.00001, Val_SpeedRefEUMax := 130.0, Val_SpeedFdbkEUMax := 130.0, SrcQ_IO := 2, SrcQ := 2, Val_Fdbk := 1, Val_Sts := 2,
        Sts_RunningFwd := 1, Sts_CommandDir := 1, Sts_ActualDir := 1, Sts_Available := 1, Sts_Prog := 1, Sts_Normal := 1, Sts_ExtReqInh := 1, Ack_FailToStart := 1, Ack_FailToStop := 1, Ack_IntlkTrip := 1, Ack_DriveFault := 1, Ack_IOFault := 1);   // TagDescript
   P1_FwdPerm : P_Perm := (Inp_Perm00 := 1, Inp_Perm01 := 1, Inp_Perm02 := 1, Inp_Perm03 := 1, Inp_Perm04 := 1, Inp_Perm05 := 1, Inp_Perm06 := 1, Inp_Perm07 := 1, Inp_Perm08 := 1, Inp_Perm09 := 1, Inp_Perm10 := 1, Inp_Perm11 := 1, Inp_Perm12 := 1, Inp_Perm13 := 1, Inp_Perm14 := 1, Inp_Perm15 := 1, Cfg_OKState := 2#1111_1111_1111_1111, Sts_PermOK := 1, Sts_NBPermOK := 1, Sts_Perm := 2#1111_1111_1111_1111);   // TagDescript - Forward Permissive
   P1_Intlk : P_Intlk := (Sts_IntlkOK := 1, Sts_NBIntlkOK := 1);   // TagDescript - Interlocks
   P1_RevPerm : P_Perm := (Inp_Perm00 := 1, Inp_Perm01 := 1, Inp_Perm02 := 1, Inp_Perm03 := 1, Inp_Perm04 := 1, Inp_Perm05 := 1, Inp_Perm06 := 1, Inp_Perm07 := 1, Inp_Perm08 := 1, Inp_Perm09 := 1, Inp_Perm10 := 1, Inp_Perm11 := 1, Inp_Perm12 := 1, Inp_Perm13 := 1, Inp_Perm14 := 1, Inp_Perm15 := 1, Cfg_OKState := 2#1111_1111_1111_1111, Sts_PermOK := 1, Sts_NBPermOK := 1, Sts_Perm := 2#1111_1111_1111_1111);   // TagDescript - Reverse Permissive
   P1_RunTime : P_RunTime := (Inp_Running := 1, Val_Starts := 9, Val_CurRunHrs := 0.8526389, Val_MaxRunHrs := 5.660138, Val_TotRunHrs := 7.8);   // TagDescript - RunTime
   PF4xx_FaultCodeList : P_DescList[36] := ([0].Desc := 'Check drive manual for this fault code', [1].Code := 71, [1].Desc := 'Network Loss', [2].Code := 81, [2].Desc := 'Communication Loss', [3].Code := 111, [3].Desc := 'Enable Hardware', [4].Code := 63, [4].Desc := 'SW OverCurrent', [5].Code := 64, [5].Desc := 'Drive Overload', [6].Code := 2, [6].Desc := 'Auxiliary Input', [7].Code := 3, [7].Desc := 'Power Loss', [8].Code := 4, [8].Desc := 'Under Voltage', [9].Code := 5, [9].Desc := 'Over Voltage', [10].Code := 6, [10].Desc := 'Motor Stalled', [11].Code := 7, [11].Desc := 'Motor Overload', [12].Code := 8, [12].Desc := 'Heatsink OverTemp', [13].Code := 12, [13].Desc := 'Hardware Overcurrent', [14].Code := 13, [14].Desc := 'Ground Fault', [15].Code := 15, [15].Desc := 'Load Loss', [16].Code := 17, [16].Desc := 'Input Phase Loss', [17].Code := 29, [17].Desc := 'Analog Input Loss', [18].Code := 32, [18].Desc := 'Fan Feedback Loss', [19].Code := 33, [19].Desc := 'Auto Restart Tries', [20].Code := 38, [20].Desc := 'Phase U to Ground', [21].Code := 39, [21].Desc := 'Phase V to Ground', [22].Code := 40, [22].Desc := 'Phase W to Ground', [23].Code := 41, [23].Desc := 'Phase U-V Short', [24].Code := 42, [24].Desc := 'Phase U-W Short', [25].Code := 43, [25].Desc := 'Phase V-W Short', [26].Code := 48, [26].Desc := 'Params Defaulted', [27].Code := 70, [27].Desc := 'Power Unit Fault', [28].Code := 80, [28].Desc := 'SVC AutoTune', [29].Code := 91, [29].Desc := 'Encoder Loss', [30].Code := 94,
        [30].Desc := 'Function Loss', [31].Code := 100, [31].Desc := 'Parameter Checksum', [32].Code := 122, [32].Desc := 'I/O Board Failure ');   // PowerFlex 4 / 40 / 400 Fault Codes and Descriptions
   PF525_FaultCodeList : P_DescList[61] := ([0].Desc := 'Check drive manual for this fault code', [1].Code := 71, [1].Desc := 'DSI Net Loss', [2].Code := 72, [2].Desc := 'Opt Net Loss', [3].Code := 81, [3].Desc := 'DSI Comm Loss', [4].Code := 82, [4].Desc := 'Opt Comm Loss', [5].Code := 73, [5].Desc := 'Ethernet Net Loss', [6].Code := 83, [6].Desc := 'Ethernet Comm Loss', [7].Code := 111, [7].Desc := 'Safety Hardware', [8].Code := 59, [8].Desc := 'Safety Open', [9].Code := 63, [9].Desc := 'SW Over Current', [10].Code := 64, [10].Desc := 'Drive Overload', [11].Code := 2, [11].Desc := 'Auxiliary Input', [12].Code := 3, [12].Desc := 'Power Loss', [13].Code := 4, [13].Desc := 'Under Voltage', [14].Code := 5, [14].Desc := 'Over Voltage', [15].Code := 6, [15].Desc := 'Motor Stalled', [16].Code := 7, [16].Desc := 'Motor Overload', [17].Code := 8, [17].Desc := 'Heatsink Overtemp', [18].Code := 9, [18].Desc := 'CC OverTemp', [19].Code := 80, [19].Desc := 'AutoTune Failure', [20].Code := 12, [20].Desc := 'Hardware Overcurrent', [21].Code := 13, [21].Desc := 'Ground Fault', [22].Code := 15, [22].Desc := 'Load Loss', [23].Code := 21, [23].Desc := 'Output Phase Loss', [24].Code := 29, [24].Desc := 'Analog Input Loss', [25].Code := 33, [25].Desc := 'Auto Restart Tries', [26].Code := 38, [26].Desc := 'Phase U to Ground', [27].Code := 39, [27].Desc := 'Phase V to Ground', [28].Code := 40, [28].Desc := 'Phase W to Ground', [29].Code := 41, [29].Desc := 'Phase U-V Short', [30].Code := 42,
        [30].Desc := 'Phase U-W Short', [31].Code := 43, [31].Desc := 'Phase V-W Short', [32].Code := 70, [32].Desc := 'Power Unit', [33].Code := 91, [33].Desc := 'Encoder Loss', [34].Code := 94, [34].Desc := 'Function Loss', [35].Code := 100, [35].Desc := 'Parameter Checksum', [36].Code := 101, [36].Desc := 'External Storage', [37].Code := 105, [37].Desc := 'C Connect Error', [38].Code := 106, [38].Desc := 'Incompat. C-P', [39].Code := 107, [39].Desc := 'Replaced C-P', [40].Code := 109, [40].Desc := 'Mismatch C-P', [41].Code := 110, [41].Desc := 'Keypad Membrane', [42].Code := 48, [42].Desc := 'Parameters Defaulted', [43].Code := 114, [43].Desc := 'uC Failure', [44].Code := 122, [44].Desc := 'I/O Baord Fail', [45].Code := 125, [45].Desc := 'Flash Update Reqd', [46].Code := 126, [46].Desc := 'Unrecoverable Error', [47].Code := 127, [47].Desc := 'DSI Flash Update Reqd');   // PowerFlex 525 VFD Fault Codes and Descriptions
   PF6000_FW5_FaultCodeList : P_DescList[490] := ([0].Desc := 'Check drive manual for this fault code', [1].Code := -1, [1].Desc := 'No more fault information found', [2].Code := 654, [2].Desc := 'DCS Communication Fault', [3].Code := 655, [3].Desc := 'DCS Communication Fault Warn', [4].Code := 641, [4].Desc := 'Input Circuit Breaker Tripped', [5].Code := 642, [5].Desc := 'Transformer Over Temperature Trip', [6].Code := 643, [6].Desc := 'Transformer Over Temperature Warn', [7].Code := 644, [7].Desc := 'Power Module Cabinet Fan Fault', [8].Code := 645, [8].Desc := 'Power Module Cabinet Fan CB Open', [9].Code := 646, [9].Desc := 'Transformer Cabinet Fan Fault', [10].Code := 647, [10].Desc := 'Transformer Cabinet Fan CB Open', [11].Code := 648, [11].Desc := 'Auxiliary Power Off', [12].Code := 649, [12].Desc := 'Cabinet Door Open', [13].Code := 650, [13].Desc := 'Control Power Switch Warn', [14].Code := 651, [14].Desc := 'Analog Loss Warn', [15].Code := 652, [15].Desc := 'DSP Communication Fault', [16].Code := 653, [16].Desc := 'Cooling Fan Contactor Open', [17].Code := 656, [17].Desc := 'Feedback Analog Loss Warning', [18].Code := 433, [18].Desc := 'Output Short Circuit', [19].Code := 434, [19].Desc := 'Output Over Current', [20].Code := 435, [20].Desc := 'Motor Over Temperature', [21].Code := 436, [21].Desc := 'Output Over Voltage', [22].Code := 437, [22].Desc := 'Abnormal Output Voltage', [23].Code := 438, [23].Desc := 'Ground Fault', [24].Code := 439, [24].Desc := 'Over Speed Fault', [25].Code := 440, [25].Desc := 'Motor Stalled', [26].Code := 442, [26].Desc := 'Output Phase Over Current', [27].Code := 449, [27].Desc := 'Motor Over Temperature Warn', [28].Code := 450, [28].Desc := 'Abnormal Output Voltage Warn', [29].Code := 451, [29].Desc := 'Ground Fault Warn', [30].Code := 452,
        [30].Desc := 'Output Frequency Deviation Warn', [31].Code := 454, [31].Desc := 'Input Power Loss, Waiting For Recovery', [32].Code := 455, [32].Desc := 'Input Voltage Sag, Derating Operating', [33].Code := 456, [33].Desc := 'Low Voltage Ride Through Operating', [34].Code := 457, [34].Desc := 'Input Voltage Sag, Flux Controlling', [35].Code := 458, [35].Desc := 'Lower Ver., No PowerCell Bypass Function', [36].Code := 459, [36].Desc := 'Bypass Operating', [37].Code := 465, [37].Desc := 'Cabinet Door Open While Drive Energized', [38].Code := 466, [38].Desc := 'E-Stop Trip', [39].Code := 467, [39].Desc := 'Input CB Open (Not Initiated by Drive)', [40].Code := 468, [40].Desc := 'Non-Zero Frequency Command Upon Start', [41].Code := 469, [41].Desc := 'Flying Start Failed', [42].Code := 474, [42].Desc := 'System Locked', [43].Code := 475, [43].Desc := 'CPU Board In Wrong Position', [44].Code := 476, [44].Desc := 'AT Board In Wrong Position', [45].Code := 477, [45].Desc := '5V Power Supply Fault', [46].Code := 478, [46].Desc := '15V Power Supply Fault', [47].Code := 479, [47].Desc := '24V DCS Power Supply Fault', [48].Code := 480, [48].Desc := '24V PLC Power Supply Fault', [49].Code := 481, [49].Desc := 'PWMA Board In Wrong Position', [50].Code := 482, [50].Desc := 'PWMB Board In Wrong Position', [51].Code := 483, [51].Desc := 'PWMC Board In Wrong Position', [52].Code := 484, [52].Desc := 'DT Board In Wrong Position', [53].Code := 486, [53].Desc := 'Low Voltage Ride Through Over Time Limit', [54].Code := 487, [54].Desc := 'Low Voltage Ride Through Short Interval ', [55].Code := 488, [55].Desc := 'Low Voltage Ride Through Failure', [56].Code := 489, [56].Desc := 'Input Voltage Loss While Stop', [57].Code := 490, [57].Desc := 'Input Voltage Loss Over Time Limit', [58].Code := 492, [58].Desc := 'Input Voltage Loss', [59].Code := 493, [59].Desc := 'Bypass Over Time Limit', [60].Code := 494,
        [60].Desc := 'Bypass Start Failure', [61].Code := 561, [61].Desc := 'Overtemp Time Out In Power Cell #1', [62].Code := 562, [62].Desc := 'Overtemp Time Out In Power Cell #2', [63].Code := 563, [63].Desc := 'Overtemp Time Out In Power Cell #3', [64].Code := 564, [64].Desc := 'Overtemp Time Out In Power Cell #4', [65].Code := 565, [65].Desc := 'Overtemp Time Out In Power Cell #5', [66].Code := 566, [66].Desc := 'Overtemp Time Out In Power Cell #6', [67].Code := 567, [67].Desc := 'Overtemp Time Out In Power Cell #7', [68].Code := 568, [68].Desc := 'Overtemp Time Out In Power Cell #8', [69].Code := 569, [69].Desc := 'Overtemp Time Out In Power Cell #9', [70].Code := 570, [70].Desc := 'Overtemp Time Out In Power Cell #10', [71].Code := 571, [71].Desc := 'Overtemp Time Out In Power Cell #11', [72].Code := 572, [72].Desc := 'Overtemp Time Out In Power Cell #12', [73].Code := 573, [73].Desc := 'Overtemp Time Out In Power Cell #13', [74].Code := 574, [74].Desc := 'Overtemp Time Out In Power Cell #14', [75].Code := 575, [75].Desc := 'Overtemp Time Out In Power Cell #15', [76].Code := 576, [76].Desc := 'Overtemp Time Out In Power Cell #16', [77].Code := 577, [77].Desc := 'Overtemp Time Out In Power Cell #17', [78].Code := 578, [78].Desc := 'Overtemp Time Out In Power Cell #18', [79].Code := 579, [79].Desc := 'Overtemp Time Out In Power Cell #19', [80].Code := 580, [80].Desc := 'Overtemp Time Out In Power Cell #20', [81].Code := 581, [81].Desc := 'Overtemp Time Out In Power Cell #21', [82].Code := 582, [82].Desc := 'Overtemp Time Out In Power Cell #22', [83].Code := 583, [83].Desc := 'Overtemp Time Out In Power Cell #23', [84].Code := 584, [84].Desc := 'Overtemp Time Out In Power Cell #24', [85].Code := 585, [85].Desc := 'Overtemp Time Out In Power Cell #25', [86].Code := 586, [86].Desc := 'Overtemp Time Out In Power Cell #26', [87].Code := 587, [87].Desc := 'Overtemp Time Out In Power Cell #27', [88].Code := 1, [88].Desc := 'IGBT Over Current In Power Cell #1', [89].Code := 2, [89].Desc := 'Capacitor Abnormal In Power Cell #1', [90].Code := 3,
        [90].Desc := 'Input Over Voltage In Power Cell #1', [91].Code := 4, [91].Desc := 'DCBus Undervolt In Power Cell #1 Warn', [92].Code := 5, [92].Desc := 'Communication Error In Power Cell #1', [93].Code := 6, [93].Desc := 'No PWM Pulse For IGBT In Power cell #1', [94].Code := 9, [94].Desc := 'IGBT Failed To Turn On In Power Cell #1', [95].Code := 10, [95].Desc := 'Power Cell #1 Bypassed', [96].Code := 11, [96].Desc := 'Over Temperature In Power Cell #1', [97].Code := 12, [97].Desc := 'Power Cell #1 Failed To Bypass', [98].Code := 13, [98].Desc := 'One Phase Lost In Power Cell #1', [99].Code := 14, [99].Desc := 'Two Phases Lost In Power Cell #1', [100].Code := 15, [100].Desc := 'Bypass Failure (OV) In Power Cell #1', [101].Code := 17, [101].Desc := 'IGBT Over Current In Power Cell #2', [102].Code := 18, [102].Desc := 'Capacitor Abnormal In Power Cell #2', [103].Code := 19, [103].Desc := 'Input Over Voltage In Power Cell #2', [104].Code := 20, [104].Desc := 'DCBus Undervolt In Power Cell #2 Warn', [105].Code := 21, [105].Desc := 'Communication Error In Power Cell #2', [106].Code := 22, [106].Desc := 'No PWM Pulse For IGBT In Power cell #2', [107].Code := 25, [107].Desc := 'IGBT Failed To Turn On In Power Cell #2', [108].Code := 26, [108].Desc := 'Power Cell #2 Bypassed', [109].Code := 27, [109].Desc := 'Over Temperature In Power Cell #2', [110].Code := 28, [110].Desc := 'Power Cell #2 Failed To Bypass', [111].Code := 29, [111].Desc := 'One Phase Lost In Power Cell #2', [112].Code := 30, [112].Desc := 'Two Phases Lost In Power Cell #2', [113].Code := 31, [113].Desc := 'Bypass Failure (OV) In Power Cell #2', [114].Code := 33, [114].Desc := 'IGBT Over Current In Power Cell #3', [115].Code := 34, [115].Desc := 'Capacitor Abnormal In Power Cell #3', [116].Code := 35, [116].Desc := 'Input Over Voltage In Power Cell #3', [117].Code := 36, [117].Desc := 'DCBus Undervolt In Power Cell #3 Warn', [118].Code := 37, [118].Desc := 'Communication Error In Power Cell #3', [119].Code := 38, [119].Desc := 'No PWM Pulse For IGBT In Power cell #3', [120].Code := 41,
        [120].Desc := 'IGBT Failed To Turn On In Power Cell #3', [121].Code := 42, [121].Desc := 'Power Cell #3 Bypassed', [122].Code := 43, [122].Desc := 'Over Temperature In Power Cell #3', [123].Code := 44, [123].Desc := 'Power Cell #3 Failed To Bypass', [124].Code := 45, [124].Desc := 'One Phase Lost In Power Cell #3', [125].Code := 46, [125].Desc := 'Two Phases Lost In Power Cell #3', [126].Code := 47, [126].Desc := 'Bypass Failure (OV) In Power Cell #3', [127].Code := 49, [127].Desc := 'IGBT Over Current In Power Cell #4', [128].Code := 50, [128].Desc := 'Capacitor Abnormal In Power Cell #4', [129].Code := 51, [129].Desc := 'Input Over Voltage In Power Cell #4', [130].Code := 52, [130].Desc := 'DCBus Undervolt In Power Cell #4 Warn', [131].Code := 53, [131].Desc := 'Communication Error In Power Cell #4', [132].Code := 54, [132].Desc := 'No PWM Pulse For IGBT In Power cell #4', [133].Code := 57, [133].Desc := 'IGBT Failed To Turn On In Power Cell #4', [134].Code := 58, [134].Desc := 'Power Cell #4 Bypassed', [135].Code := 59, [135].Desc := 'Over Temperature In Power Cell #4', [136].Code := 60, [136].Desc := 'Power Cell #4 Failed To Bypass', [137].Code := 61, [137].Desc := 'One Phase Lost In Power Cell #4', [138].Code := 62, [138].Desc := 'Two Phases Lost In Power Cell #4', [139].Code := 63, [139].Desc := 'Bypass Failure (OV) In Power Cell #4', [140].Code := 65, [140].Desc := 'IGBT Over Current In Power Cell #5', [141].Code := 66, [141].Desc := 'Capacitor Abnormal In Power Cell #5', [142].Code := 67, [142].Desc := 'Input Over Voltage In Power Cell #5', [143].Code := 68, [143].Desc := 'DCBus Undervolt In Power Cell #5 Warn', [144].Code := 69, [144].Desc := 'Communication Error In Power Cell #5', [145].Code := 70, [145].Desc := 'No PWM Pulse For IGBT In Power cell #5', [146].Code := 73, [146].Desc := 'IGBT Failed To Turn On In Power Cell #5', [147].Code := 74, [147].Desc := 'Power Cell #5 Bypassed', [148].Code := 75, [148].Desc := 'Over Temperature In Power Cell #5', [149].Code := 76, [149].Desc := 'Power Cell #5 Failed To Bypass', [150].Code := 77,
        [150].Desc := 'One Phase Lost In Power Cell #5', [151].Code := 78, [151].Desc := 'Two Phases Lost In Power Cell #5', [152].Code := 79, [152].Desc := 'Bypass Failure (OV) In Power Cell #5', [153].Code := 81, [153].Desc := 'IGBT Over Current In Power Cell #6', [154].Code := 82, [154].Desc := 'Capacitor Abnormal In Power Cell #6', [155].Code := 83, [155].Desc := 'Input Over Voltage In Power Cell #6', [156].Code := 84, [156].Desc := 'DCBus Undervolt In Power Cell #6 Warn', [157].Code := 85, [157].Desc := 'Communication Error In Power Cell #6', [158].Code := 86, [158].Desc := 'No PWM Pulse For IGBT In Power cell #6', [159].Code := 89, [159].Desc := 'IGBT Failed To Turn On In Power Cell #6', [160].Code := 90, [160].Desc := 'Power Cell #6 Bypassed', [161].Code := 91, [161].Desc := 'Over Temperature In Power Cell #6', [162].Code := 92, [162].Desc := 'Power Cell #6 Failed To Bypass', [163].Code := 93, [163].Desc := 'One Phase Lost In Power Cell #6', [164].Code := 94, [164].Desc := 'Two Phases Lost In Power Cell #6', [165].Code := 95, [165].Desc := 'Bypass Failure (OV) In Power Cell #6', [166].Code := 97, [166].Desc := 'IGBT Over Current In Power Cell #7', [167].Code := 98, [167].Desc := 'Capacitor Abnormal In Power Cell #7', [168].Code := 99, [168].Desc := 'Input Over Voltage In Power Cell #7', [169].Code := 100, [169].Desc := 'DCBus Undervolt In Power Cell #7 Warn', [170].Code := 101, [170].Desc := 'Communication Error In Power Cell #7', [171].Code := 102, [171].Desc := 'No PWM Pulse For IGBT In Power cell #7', [172].Code := 105, [172].Desc := 'IGBT Failed To Turn On In Power Cell #7', [173].Code := 106, [173].Desc := 'Power Cell #7 Bypassed', [174].Code := 107, [174].Desc := 'Over Temperature In Power Cell #7', [175].Code := 108, [175].Desc := 'Power Cell #7 Failed To Bypass', [176].Code := 109, [176].Desc := 'One Phase Lost In Power Cell #7', [177].Code := 110, [177].Desc := 'Two Phases Lost In Power Cell #7', [178].Code := 111, [178].Desc := 'Bypass Failure (OV) In Power Cell #7', [179].Code := 113, [179].Desc := 'IGBT Over Current In Power Cell #8', [180].Code := 114,
        [180].Desc := 'Capacitor Abnormal In Power Cell #8', [181].Code := 115, [181].Desc := 'Input Over Voltage In Power Cell #8', [182].Code := 116, [182].Desc := 'DCBus Undervolt In Power Cell #8 Warn', [183].Code := 117, [183].Desc := 'Communication Error In Power Cell #8', [184].Code := 118, [184].Desc := 'No PWM Pulse For IGBT In Power cell #8', [185].Code := 121, [185].Desc := 'IGBT Failed To Turn On In Power Cell #8', [186].Code := 122, [186].Desc := 'Power Cell #8 Bypassed', [187].Code := 123, [187].Desc := 'Over Temperature In Power Cell #8', [188].Code := 124, [188].Desc := 'Power Cell #8 Failed To Bypass', [189].Code := 125, [189].Desc := 'One Phase Lost In Power Cell #8', [190].Code := 126, [190].Desc := 'Two Phases Lost In Power Cell #8', [191].Code := 127, [191].Desc := 'Bypass Failure (OV) In Power Cell #8', [192].Code := 129, [192].Desc := 'IGBT Over Current In Power Cell #9', [193].Code := 130, [193].Desc := 'Capacitor Abnormal In Power Cell #9', [194].Code := 131, [194].Desc := 'Input Over Voltage In Power Cell #9', [195].Code := 132, [195].Desc := 'DCBus Undervolt In Power Cell #9 Warn', [196].Code := 133, [196].Desc := 'Communication Error In Power Cell #9', [197].Code := 134, [197].Desc := 'No PWM Pulse For IGBT In Power cell #9', [198].Code := 137, [198].Desc := 'IGBT Failed To Turn On In Power Cell #9', [199].Code := 138, [199].Desc := 'Power Cell #9 Bypassed', [200].Code := 139, [200].Desc := 'Over Temperature In Power Cell #9', [201].Code := 140, [201].Desc := 'Power Cell #9 Failed To Bypass', [202].Code := 141, [202].Desc := 'One Phase Lost In Power Cell #9', [203].Code := 142, [203].Desc := 'Two Phases Lost In Power Cell #9', [204].Code := 143, [204].Desc := 'Bypass Failure (OV) In Power Cell #9', [205].Code := 145, [205].Desc := 'IGBT Over Current In Power Cell #10', [206].Code := 146, [206].Desc := 'Capacitor Abnormal In Power Cell #10', [207].Code := 147, [207].Desc := 'Input Over Voltage In Power Cell #10', [208].Code := 148, [208].Desc := 'DCBus Undervolt In Power Cell #10 Warn', [209].Code := 149, [209].Desc := 'Communication Error In Power Cell #10', [210].Code := 150,
        [210].Desc := 'No PWM Pulse For IGBT In Power cell #10', [211].Code := 153, [211].Desc := 'IGBT Failed To Turn On In Power Cell #10', [212].Code := 154, [212].Desc := 'Power Cell #10 Bypassed', [213].Code := 155, [213].Desc := 'Over Temperature In Power Cell #10', [214].Code := 156, [214].Desc := 'Power Cell #10 Failed To Bypass', [215].Code := 157, [215].Desc := 'One Phase Lost In Power Cell #10', [216].Code := 158, [216].Desc := 'Two Phases Lost In Power Cell #10', [217].Code := 159, [217].Desc := 'Bypass Failure (OV) In Power Cell #10', [218].Code := 161, [218].Desc := 'IGBT Over Current In Power Cell #11', [219].Code := 162, [219].Desc := 'Capacitor Abnormal In Power Cell #11', [220].Code := 163, [220].Desc := 'Input Over Voltage In Power Cell #11', [221].Code := 164, [221].Desc := 'DCBus Undervolt In Power Cell #11 Warn', [222].Code := 165, [222].Desc := 'Communication Error In Power Cell #11', [223].Code := 166, [223].Desc := 'No PWM Pulse For IGBT In Power cell #11', [224].Code := 169, [224].Desc := 'IGBT Failed To Turn On In Power Cell #11', [225].Code := 170, [225].Desc := 'Power Cell #11 Bypassed', [226].Code := 171, [226].Desc := 'Over Temperature In Power Cell #11', [227].Code := 172, [227].Desc := 'Power Cell #11 Failed To Bypass', [228].Code := 173, [228].Desc := 'One Phase Lost In Power Cell #11', [229].Code := 174, [229].Desc := 'Two Phases Lost In Power Cell #11', [230].Code := 175, [230].Desc := 'Bypass Failure (OV) In Power Cell #11', [231].Code := 177, [231].Desc := 'IGBT Over Current In Power Cell #12', [232].Code := 178, [232].Desc := 'Capacitor Abnormal In Power Cell #12', [233].Code := 179, [233].Desc := 'Input Over Voltage In Power Cell #12', [234].Code := 180, [234].Desc := 'DCBus Undervolt In Power Cell #12 Warn', [235].Code := 181, [235].Desc := 'Communication Error In Power Cell #12', [236].Code := 182, [236].Desc := 'No PWM Pulse For IGBT In Power cell #12', [237].Code := 185, [237].Desc := 'IGBT Failed To Turn On In Power Cell #12', [238].Code := 186, [238].Desc := 'Power Cell #12 Bypassed', [239].Code := 187, [239].Desc := 'Over Temperature In Power Cell #12', [240].Code := 188,
        [240].Desc := 'Power Cell #12 Failed To Bypass', [241].Code := 189, [241].Desc := 'One Phase Lost In Power Cell #12', [242].Code := 190, [242].Desc := 'Two Phases Lost In Power Cell #12', [243].Code := 191, [243].Desc := 'Bypass Failure (OV) In Power Cell #12', [244].Code := 193, [244].Desc := 'IGBT Over Current In Power Cell #13', [245].Code := 194, [245].Desc := 'Capacitor Abnormal In Power Cell #13', [246].Code := 195, [246].Desc := 'Input Over Voltage In Power Cell #13', [247].Code := 196, [247].Desc := 'DCBus Undervolt In Power Cell #13 Warn', [248].Code := 197, [248].Desc := 'Communication Error In Power Cell #13', [249].Code := 198, [249].Desc := 'No PWM Pulse For IGBT In Power cell #13', [250].Code := 201, [250].Desc := 'IGBT Failed To Turn On In Power Cell #13', [251].Code := 202, [251].Desc := 'Power Cell #13 Bypassed', [252].Code := 203, [252].Desc := 'Over Temperature In Power Cell #13', [253].Code := 204, [253].Desc := 'Power Cell #13 Failed To Bypass', [254].Code := 205, [254].Desc := 'One Phase Lost In Power Cell #13', [255].Code := 206, [255].Desc := 'Two Phases Lost In Power Cell #13', [256].Code := 207, [256].Desc := 'Bypass Failure (OV) In Power Cell #13', [257].Code := 209, [257].Desc := 'IGBT Over Current In Power Cell #14', [258].Code := 210, [258].Desc := 'Capacitor Abnormal In Power Cell #14', [259].Code := 211, [259].Desc := 'Input Over Voltage In Power Cell #14', [260].Code := 212, [260].Desc := 'DCBus Undervolt In Power Cell #14 Warn', [261].Code := 213, [261].Desc := 'Communication Error In Power Cell #14', [262].Code := 214, [262].Desc := 'No PWM Pulse For IGBT In Power cell #14', [263].Code := 217, [263].Desc := 'IGBT Failed To Turn On In Power Cell #14', [264].Code := 218, [264].Desc := 'Power Cell #14 Bypassed', [265].Code := 219, [265].Desc := 'Over Temperature In Power Cell #14', [266].Code := 220, [266].Desc := 'Power Cell #14 Failed To Bypass', [267].Code := 221, [267].Desc := 'One Phase Lost In Power Cell #14', [268].Code := 222, [268].Desc := 'Two Phases Lost In Power Cell #14', [269].Code := 223, [269].Desc := 'Bypass Failure (OV) In Power Cell #14', [270].Code := 225,
        [270].Desc := 'IGBT Over Current In Power Cell #15', [271].Code := 226, [271].Desc := 'Capacitor Abnormal In Power Cell #15', [272].Code := 227, [272].Desc := 'Input Over Voltage In Power Cell #15', [273].Code := 228, [273].Desc := 'DCBus Undervolt In Power Cell #15 Warn', [274].Code := 229, [274].Desc := 'Communication Error In Power Cell #15', [275].Code := 230, [275].Desc := 'No PWM Pulse For IGBT In Power cell #15', [276].Code := 233, [276].Desc := 'IGBT Failed To Turn On In Power Cell #15', [277].Code := 234, [277].Desc := 'Power Cell #15 Bypassed', [278].Code := 235, [278].Desc := 'Over Temperature In Power Cell #15', [279].Code := 236, [279].Desc := 'Power Cell #15 Failed To Bypass', [280].Code := 237, [280].Desc := 'One Phase Lost In Power Cell #15', [281].Code := 238, [281].Desc := 'Two Phases Lost In Power Cell #15', [282].Code := 239, [282].Desc := 'Bypass Failure (OV) In Power Cell #15', [283].Code := 241, [283].Desc := 'IGBT Over Current In Power Cell #16', [284].Code := 242, [284].Desc := 'Capacitor Abnormal In Power Cell #16', [285].Code := 243, [285].Desc := 'Input Over Voltage In Power Cell #16', [286].Code := 244, [286].Desc := 'DCBus Undervolt In Power Cell #16 Warn', [287].Code := 245, [287].Desc := 'Communication Error In Power Cell #16', [288].Code := 246, [288].Desc := 'No PWM Pulse For IGBT In Power cell #16', [289].Code := 249, [289].Desc := 'IGBT Failed To Turn On In Power Cell #16', [290].Code := 250, [290].Desc := 'Power Cell #16 Bypassed', [291].Code := 251, [291].Desc := 'Over Temperature In Power Cell #16', [292].Code := 252, [292].Desc := 'Power Cell #16 Failed To Bypass', [293].Code := 253, [293].Desc := 'One Phase Lost In Power Cell #16', [294].Code := 254, [294].Desc := 'Two Phases Lost In Power Cell #16', [295].Code := 255, [295].Desc := 'Bypass Failure (OV) In Power Cell #16', [296].Code := 257, [296].Desc := 'IGBT Over Current In Power Cell #17', [297].Code := 258, [297].Desc := 'Capacitor Abnormal In Power Cell #17', [298].Code := 259, [298].Desc := 'Input Over Voltage In Power Cell #17', [299].Code := 260, [299].Desc := 'DCBus Undervolt In Power Cell #17 Warn', [300].Code := 261,
        [300].Desc := 'Communication Error In Power Cell #17', [301].Code := 262, [301].Desc := 'No PWM Pulse For IGBT In Power cell #17', [302].Code := 265, [302].Desc := 'IGBT Failed To Turn On In Power Cell #17', [303].Code := 266, [303].Desc := 'Power Cell #17 Bypassed', [304].Code := 267, [304].Desc := 'Over Temperature In Power Cell #17', [305].Code := 268, [305].Desc := 'Power Cell #17 Failed To Bypass', [306].Code := 269, [306].Desc := 'One Phase Lost In Power Cell #17', [307].Code := 270, [307].Desc := 'Two Phases Lost In Power Cell #17', [308].Code := 271, [308].Desc := 'Bypass Failure (OV) In Power Cell #17', [309].Code := 273, [309].Desc := 'IGBT Over Current In Power Cell #18', [310].Code := 274, [310].Desc := 'Capacitor Abnormal In Power Cell #18', [311].Code := 275, [311].Desc := 'Input Over Voltage In Power Cell #18', [312].Code := 276, [312].Desc := 'DCBus Undervolt In Power Cell #18 Warn', [313].Code := 277, [313].Desc := 'Communication Error In Power Cell #18', [314].Code := 278, [314].Desc := 'No PWM Pulse For IGBT In Power cell #18', [315].Code := 281, [315].Desc := 'IGBT Failed To Turn On In Power Cell #18', [316].Code := 282, [316].Desc := 'Power Cell #18 Bypassed', [317].Code := 283, [317].Desc := 'Over Temperature In Power Cell #18', [318].Code := 284, [318].Desc := 'Power Cell #18 Failed To Bypass', [319].Code := 285, [319].Desc := 'One Phase Lost In Power Cell #18', [320].Code := 286, [320].Desc := 'Two Phases Lost In Power Cell #18', [321].Code := 287, [321].Desc := 'Bypass Failure (OV) In Power Cell #18', [322].Code := 289, [322].Desc := 'IGBT Over Current In Power Cell #19', [323].Code := 290, [323].Desc := 'Capacitor Abnormal In Power Cell #19', [324].Code := 291, [324].Desc := 'Input Over Voltage In Power Cell #19', [325].Code := 292, [325].Desc := 'DCBus Undervolt In Power Cell #19 Warn', [326].Code := 293, [326].Desc := 'Communication Error In Power Cell #19', [327].Code := 294, [327].Desc := 'No PWM Pulse For IGBT In Power cell #19', [328].Code := 297, [328].Desc := 'IGBT Failed To Turn On In Power Cell #19', [329].Code := 298, [329].Desc := 'Power Cell #19 Bypassed', [330].Code := 299,
        [330].Desc := 'Over Temperature In Power Cell #19', [331].Code := 300, [331].Desc := 'Power Cell #19 Failed To Bypass', [332].Code := 301, [332].Desc := 'One Phase Lost In Power Cell #19', [333].Code := 302, [333].Desc := 'Two Phases Lost In Power Cell #19', [334].Code := 303, [334].Desc := 'Bypass Failure (OV) In Power Cell #19', [335].Code := 305, [335].Desc := 'IGBT Over Current In Power Cell #20', [336].Code := 306, [336].Desc := 'Capacitor Abnormal In Power Cell #20', [337].Code := 307, [337].Desc := 'Input Over Voltage In Power Cell #20', [338].Code := 308, [338].Desc := 'DCBus Undervolt In Power Cell #20 Warn', [339].Code := 309, [339].Desc := 'Communication Error In Power Cell #20', [340].Code := 310, [340].Desc := 'No PWM Pulse For IGBT In Power cell #20', [341].Code := 313, [341].Desc := 'IGBT Failed To Turn On In Power Cell #20', [342].Code := 314, [342].Desc := 'Power Cell #20 Bypassed', [343].Code := 315, [343].Desc := 'Over Temperature In Power Cell #20', [344].Code := 316, [344].Desc := 'Power Cell #20 Failed To Bypass', [345].Code := 317, [345].Desc := 'One Phase Lost In Power Cell #20', [346].Code := 318, [346].Desc := 'Two Phases Lost In Power Cell #20', [347].Code := 319, [347].Desc := 'Bypass Failure (OV) In Power Cell #20', [348].Code := 321, [348].Desc := 'IGBT Over Current In Power Cell #21', [349].Code := 322, [349].Desc := 'Capacitor Abnormal In Power Cell #21', [350].Code := 323, [350].Desc := 'Input Over Voltage In Power Cell #21', [351].Code := 324, [351].Desc := 'DCBus Undervolt In Power Cell #21 Warn', [352].Code := 325, [352].Desc := 'Communication Error In Power Cell #21', [353].Code := 326, [353].Desc := 'No PWM Pulse For IGBT In Power cell #21', [354].Code := 329, [354].Desc := 'IGBT Failed To Turn On In Power Cell #21', [355].Code := 330, [355].Desc := 'Power Cell #21 Bypassed', [356].Code := 331, [356].Desc := 'Over Temperature In Power Cell #21', [357].Code := 332, [357].Desc := 'Power Cell #21 Failed To Bypass', [358].Code := 333, [358].Desc := 'One Phase Lost In Power Cell #21', [359].Code := 334, [359].Desc := 'Two Phases Lost In Power Cell #21', [360].Code := 335,
        [360].Desc := 'Bypass Failure (OV) In Power Cell #21', [361].Code := 337, [361].Desc := 'IGBT Over Current In Power Cell #22', [362].Code := 338, [362].Desc := 'Capacitor Abnormal In Power Cell #22', [363].Code := 339, [363].Desc := 'Input Over Voltage In Power Cell #22', [364].Code := 340, [364].Desc := 'DCBus Undervolt In Power Cell #22 Warn', [365].Code := 341, [365].Desc := 'Communication Error In Power Cell #22', [366].Code := 342, [366].Desc := 'No PWM Pulse For IGBT In Power cell #22', [367].Code := 345, [367].Desc := 'IGBT Failed To Turn On In Power Cell #22', [368].Code := 346, [368].Desc := 'Power Cell #22 Bypassed', [369].Code := 347, [369].Desc := 'Over Temperature In Power Cell #22', [370].Code := 348, [370].Desc := 'Power Cell #22 Failed To Bypass', [371].Code := 349, [371].Desc := 'One Phase Lost In Power Cell #22', [372].Code := 350, [372].Desc := 'Two Phases Lost In Power Cell #22', [373].Code := 351, [373].Desc := 'Bypass Failure (OV) In Power Cell #22', [374].Code := 353, [374].Desc := 'IGBT Over Current In Power Cell #23', [375].Code := 354, [375].Desc := 'Capacitor Abnormal In Power Cell #23', [376].Code := 355, [376].Desc := 'Input Over Voltage In Power Cell #23', [377].Code := 356, [377].Desc := 'DCBus Undervolt In Power Cell #23 Warn', [378].Code := 357, [378].Desc := 'Communication Error In Power Cell #23', [379].Code := 358, [379].Desc := 'No PWM Pulse For IGBT In Power cell #23', [380].Code := 361, [380].Desc := 'IGBT Failed To Turn On In Power Cell #23', [381].Code := 362, [381].Desc := 'Power Cell #23 Bypassed', [382].Code := 363, [382].Desc := 'Over Temperature In Power Cell #23', [383].Code := 364, [383].Desc := 'Power Cell #23 Failed To Bypass', [384].Code := 365, [384].Desc := 'One Phase Lost In Power Cell #23', [385].Code := 366, [385].Desc := 'Two Phases Lost In Power Cell #23', [386].Code := 367, [386].Desc := 'Bypass Failure (OV) In Power Cell #23', [387].Code := 369, [387].Desc := 'IGBT Over Current In Power Cell #24', [388].Code := 370, [388].Desc := 'Capacitor Abnormal In Power Cell #24', [389].Code := 371, [389].Desc := 'Input Over Voltage In Power Cell #24', [390].Code := 372,
        [390].Desc := 'DCBus Undervolt In Power Cell #24 Warn', [391].Code := 373, [391].Desc := 'Communication Error In Power Cell #24', [392].Code := 374, [392].Desc := 'No PWM Pulse For IGBT In Power cell #24', [393].Code := 377, [393].Desc := 'IGBT Failed To Turn On In Power Cell #24', [394].Code := 378, [394].Desc := 'Power Cell #24 Bypassed', [395].Code := 379, [395].Desc := 'Over Temperature In Power Cell #24', [396].Code := 380, [396].Desc := 'Power Cell #24 Failed To Bypass', [397].Code := 381, [397].Desc := 'One Phase Lost In Power Cell #24', [398].Code := 382, [398].Desc := 'Two Phases Lost In Power Cell #24', [399].Code := 383, [399].Desc := 'Bypass Failure (OV) In Power Cell #24', [400].Code := 385, [400].Desc := 'IGBT Over Current In Power Cell #25', [401].Code := 386, [401].Desc := 'Capacitor Abnormal In Power Cell #25', [402].Code := 387, [402].Desc := 'Input Over Voltage In Power Cell #25', [403].Code := 388, [403].Desc := 'DCBus Undervolt In Power Cell #25 Warn', [404].Code := 389, [404].Desc := 'Communication Error In Power Cell #25', [405].Code := 390, [405].Desc := 'No PWM Pulse For IGBT In Power cell #25', [406].Code := 393, [406].Desc := 'IGBT Failed To Turn On In Power Cell #25', [407].Code := 394, [407].Desc := 'Power Cell #25 Bypassed', [408].Code := 395, [408].Desc := 'Over Temperature In Power Cell #25', [409].Code := 396, [409].Desc := 'Power Cell #25 Failed To Bypass', [410].Code := 397, [410].Desc := 'One Phase Lost In Power Cell #25', [411].Code := 398, [411].Desc := 'Two Phases Lost In Power Cell #25', [412].Code := 399, [412].Desc := 'Bypass Failure (OV) In Power Cell #25', [413].Code := 401, [413].Desc := 'IGBT Over Current In Power Cell #26', [414].Code := 402, [414].Desc := 'Capacitor Abnormal In Power Cell #26', [415].Code := 403, [415].Desc := 'Input Over Voltage In Power Cell #26', [416].Code := 404, [416].Desc := 'DCBus Undervolt In Power Cell #26 Warn', [417].Code := 405, [417].Desc := 'Communication Error In Power Cell #26', [418].Code := 406, [418].Desc := 'No PWM Pulse For IGBT In Power cell #26', [419].Code := 409, [419].Desc := 'IGBT Failed To Turn On In Power Cell #26', [420].Code := 410,
        [420].Desc := 'Power Cell #26 Bypassed', [421].Code := 411, [421].Desc := 'Over Temperature In Power Cell #26', [422].Code := 412, [422].Desc := 'Power Cell #26 Failed To Bypass', [423].Code := 413, [423].Desc := 'One Phase Lost In Power Cell #26', [424].Code := 414, [424].Desc := 'Two Phases Lost In Power Cell #26', [425].Code := 415, [425].Desc := 'Bypass Failure (OV) In Power Cell #26', [426].Code := 417, [426].Desc := 'IGBT Over Current In Power Cell #27', [427].Code := 418, [427].Desc := 'Capacitor Abnormal In Power Cell #27', [428].Code := 419, [428].Desc := 'Input Over Voltage In Power Cell #27', [429].Code := 420, [429].Desc := 'DCBus Undervolt In Power Cell #27 Warn', [430].Code := 421, [430].Desc := 'Communication Error In Power Cell #27', [431].Code := 422, [431].Desc := 'No PWM Pulse For IGBT In Power cell #27', [432].Code := 425, [432].Desc := 'IGBT Failed To Turn On In Power Cell #27', [433].Code := 426, [433].Desc := 'Power Cell #27 Bypassed', [434].Code := 427, [434].Desc := 'Over Temperature In Power Cell #27', [435].Code := 428, [435].Desc := 'Power Cell #27 Failed To Bypass', [436].Code := 429, [436].Desc := 'One Phase Lost In Power Cell #27', [437].Code := 430, [437].Desc := 'Two Phases Lost In Power Cell #27', [438].Code := 431, [438].Desc := 'Bypass Failure (OV) In Power Cell #27', [439].Code := 497, [439].Desc := 'PWMA Board Incompatible With PUA1 Board', [440].Code := 498, [440].Desc := 'PWMA Board Incompatible With PUA2 Board', [441].Code := 499, [441].Desc := 'PWMA Board Incompatible With PUA3 Board', [442].Code := 500, [442].Desc := 'PWMA Board Incompatible With PUA4 Board', [443].Code := 501, [443].Desc := 'PWMA Board Incompatible With PUA5 Board', [444].Code := 502, [444].Desc := 'PWMA Board Incompatible With PUA6 Board', [445].Code := 503, [445].Desc := 'PWMA Board Incompatible With PUA7 Board', [446].Code := 504, [446].Desc := 'PWMA Board Incompatible With PUA8 Board', [447].Code := 505, [447].Desc := 'PWMA Board Incompatible With PUA9 Board', [448].Code := 506, [448].Desc := 'PWMA Board Incompatible With PUA10 Board', [449].Code := 507, [449].Desc := 'PWMA Board Incompatible With PUA11 Board', [450].Code := 508,
        [450].Desc := 'PWMA Board Incompatible With PUA12 Board', [451].Code := 509, [451].Desc := 'PWMA Board Incompatible With PUA13 Board', [452].Code := 510, [452].Desc := 'Pri. FPGA Incompatible With PWMA Board', [453].Code := 511, [453].Desc := 'Pri. FPGA Incompatible With PWMB Board', [454].Code := 512, [454].Desc := 'Pri. FPGA Incompatible With PWMC Board', [455].Code := 513, [455].Desc := 'PWMB Board Incompatible With PUB1 Board', [456].Code := 514, [456].Desc := 'PWMB Board Incompatible With PUB2 Board', [457].Code := 515, [457].Desc := 'PWMB Board Incompatible With PUB3 Board', [458].Code := 516, [458].Desc := 'PWMB Board Incompatible With PUB4 Board', [459].Code := 517, [459].Desc := 'PWMB Board Incompatible With PUB5 Board', [460].Code := 518, [460].Desc := 'PWMB Board Incompatible With PUB6 Board', [461].Code := 519, [461].Desc := 'PWMB Board Incompatible With PUB7 Board', [462].Code := 520, [462].Desc := 'PWMB Board Incompatible With PUB8 Board', [463].Code := 521, [463].Desc := 'PWMB Board Incompatible With PUB9 Board', [464].Code := 522, [464].Desc := 'PWMB Board Incompatible With PUB10 Board', [465].Code := 523, [465].Desc := 'PWMB Board Incompatible With PUB11 Board', [466].Code := 524, [466].Desc := 'PWMB Board Incompatible With PUB12 Board', [467].Code := 525, [467].Desc := 'PWMB Board Incompatible With PUB13 Board', [468].Code := 526, [468].Desc := 'Pri. FPGA Incompatible With DT Board', [469].Code := 527, [469].Desc := 'Pri. DSP Incompatible With Pri. FPGA', [470].Code := 528, [470].Desc := 'Pri. DSP Incompatible With Secondary DSP', [471].Code := 529, [471].Desc := 'PWMC Board Incompatible With PUC1 Board', [472].Code := 530, [472].Desc := 'PWMC Board Incompatible With PUC2 Board', [473].Code := 531, [473].Desc := 'PWMC Board Incompatible With PUC3 Board', [474].Code := 532, [474].Desc := 'PWMC Board Incompatible With PUC4 Board', [475].Code := 533, [475].Desc := 'PWMC Board Incompatible With PUC5 Board', [476].Code := 534, [476].Desc := 'PWMC Board Incompatible With PUC6 Board', [477].Code := 535, [477].Desc := 'PWMC Board Incompatible With PUC7 Board', [478].Code := 536, [478].Desc := 'PWMC Board Incompatible With PUC8 Board', [479].Code := 537, [479].Desc := 'PWMC Board Incompatible With PUC9 Board', [480].Code := 538,
        [480].Desc := 'PWMC Board Incompatible With PUC10 Board', [481].Code := 539, [481].Desc := 'PWMC Board Incompatible With PUC11 Board', [482].Code := 540, [482].Desc := 'PWMC Board Incompatible With PUC12 Board', [483].Code := 541, [483].Desc := 'PWMC Board Incompatible With PUC13 Board', [484].Code := 542, [484].Desc := 'Versions Of System Incompatible', [485].Code := 543, [485].Desc := 'Version Fault Identification Code Error', [486].Code := 545, [486].Desc := 'Pri. DSP Incompatible With PLC', [487].Code := 546, [487].Desc := 'HMI Incompatible With PLC', [488].Code := 547, [488].Desc := 'Pri. DSP Incompatible With HMI');   // PowerFlex 6000 MV VFD FW5.x Fault Codes and Descriptions
   PF6000_FW6_FaultCodeList : P_DescList[594] := ([0].Desc := 'Check drive manual for this fault code', [1].Code := -1, [1].Desc := 'No more fault information found', [2].Code := 654, [2].Desc := 'DCS Communication Error', [3].Code := 655, [3].Desc := 'DCS Communication Error Warning', [4].Code := 656, [4].Desc := 'Analog Feedback Loss Warning', [5].Code := 657, [5].Desc := 'Motor Over Temperature', [6].Code := 658, [6].Desc := 'Filter Cabinet Over Temperature', [7].Code := 659, [7].Desc := 'Motor Side HECS Power Supply Fault ', [8].Code := 660, [8].Desc := 'Analog Channel #2 Loss Warning', [9].Code := 433, [9].Desc := 'Motor Over Current 2', [10].Code := 434, [10].Desc := 'Motor Over Current 1', [11].Code := 435, [11].Desc := 'Fan Failure In Fan Group #1', [12].Code := 436, [12].Desc := 'Output Over Voltage', [13].Code := 437, [13].Desc := 'Abnormal Output Voltage', [14].Code := 438, [14].Desc := 'Ground Fault', [15].Code := 439, [15].Desc := 'Over Speed Fault', [16].Code := 440, [16].Desc := 'Motor Stalled', [17].Code := 442, [17].Desc := 'Output Phase Over Current', [18].Code := 443, [18].Desc := 'VFD Over Current 1', [19].Code := 444, [19].Desc := 'Fan Failure In Fan Group #2', [20].Code := 445, [20].Desc := 'Pre-Charge Contactor Failure', [21].Code := 446, [21].Desc := 'Pre-Charge Timeout', [22].Code := 447, [22].Desc := 'Pre-Charge Repeat Interval Low', [23].Code := 449, [23].Desc := 'Fan Failure Warning In Fan Group #1', [24].Code := 450, [24].Desc := 'Abnormal Output Voltage Warning', [25].Code := 451, [25].Desc := 'Ground Fault Warning', [26].Code := 452, [26].Desc := 'Output Frequency Deviation Warning', [27].Code := 454, [27].Desc := 'Input Power Loss, Waiting For Recovery', [28].Code := 455, [28].Desc := 'Input Voltage Sag, Derating Operating', [29].Code := 456, [29].Desc := 'Low Voltage Ride Through Operating', [30].Code := 457,
        [30].Desc := 'Input Voltage Sag, Flux Controlling', [31].Code := 458, [31].Desc := 'Fan Failure Warning In Fan Group #2', [32].Code := 459, [32].Desc := 'Bypass Operating', [33].Code := 460, [33].Desc := 'DC Bus Under Voltage Warning', [34].Code := 461, [34].Desc := 'Fan Failure Warning In Fan Group #3', [35].Code := 462, [35].Desc := 'Line Neutral Over Voltage Warning', [36].Code := 463, [36].Desc := 'Line Under Voltage Warning', [37].Code := 464, [37].Desc := 'Fan Failure Warning In Fan Group #4', [38].Code := 465, [38].Desc := 'Cabinet Door Open While Drive Energized', [39].Code := 466, [39].Desc := 'E-Stop Trip', [40].Code := 467, [40].Desc := 'Input Circuit Breaker Tripped', [41].Code := 468, [41].Desc := 'Non-Zero Frequency Command On Start', [42].Code := 469, [42].Desc := 'Flying Start Failed', [43].Code := 474, [43].Desc := 'System Locked', [44].Code := 475, [44].Desc := 'CPU Board In Wrong Position', [45].Code := 476, [45].Desc := 'AT Board In Wrong Position', [46].Code := 477, [46].Desc := '5V Power Supply Fault', [47].Code := 478, [47].Desc := '15V Power Supply Fault', [48].Code := 479, [48].Desc := '24V DCS Power Supply Fault', [49].Code := 480, [49].Desc := '24V PLC Power Supply Fault', [50].Code := 481, [50].Desc := 'PWMA Board In Wrong Position', [51].Code := 482, [51].Desc := 'PWMB Board In Wrong Position', [52].Code := 483, [52].Desc := 'PWMC Board In Wrong Position', [53].Code := 484, [53].Desc := 'DT Board In Wrong Position', [54].Code := 486, [54].Desc := 'Low Voltage Ride Through Over Max Time', [55].Code := 487, [55].Desc := 'Low Voltage Ride Through Short Interval', [56].Code := 488, [56].Desc := 'Low Voltage Ride Through Failure', [57].Code := 489, [57].Desc := 'Input Voltage Loss While Stop', [58].Code := 490, [58].Desc := 'Input Voltage Loss Over Time Limit', [59].Code := 492, [59].Desc := 'Input Voltage Loss', [60].Code := 493,
        [60].Desc := 'Cell Bypass Timeout', [61].Code := 494, [61].Desc := 'Cell Bypass Start Fault', [62].Code := 495, [62].Desc := 'Cell Bypass Logic Fault', [63].Code := 593, [63].Desc := 'DIP Configuration Fault In PWMA', [64].Code := 594, [64].Desc := 'Bypass Cell Re-activation Fault', [65].Code := 595, [65].Desc := 'PCCB Parameters R/W Timeout', [66].Code := 596, [66].Desc := 'Power Cells Parameters Mismatch', [67].Code := 597, [67].Desc := 'DC Bus Voltage Deviation Fault', [68].Code := 598, [68].Desc := 'DIP Configuration Fault In PWMB', [69].Code := 599, [69].Desc := 'DIP Configuration Fault In PWMC', [70].Code := 600, [70].Desc := 'Transformer Cabinet Fan Config Error', [71].Code := 609, [71].Desc := 'Line Over Voltage ', [72].Code := 610, [72].Desc := 'Line Neutral Over Voltage ', [73].Code := 611, [73].Desc := 'Line Short Circuit ', [74].Code := 612, [74].Desc := 'Line Voltage Unbalance', [75].Code := 613, [75].Desc := 'Line Current Unbalance', [76].Code := 614, [76].Desc := 'Line Side VSB Feedback Loss', [77].Code := 615, [77].Desc := 'Fan Failure In Fan Group #4', [78].Code := 616, [78].Desc := 'Pre-Charge Resistor Short Circuit', [79].Code := 617, [79].Desc := 'VFD Over Current 2', [80].Code := 618, [80].Desc := 'DC Bus Under Voltage Fault', [81].Code := 641, [81].Desc := 'Input Circuit Breaker Tripped', [82].Code := 642, [82].Desc := 'Transformer Over Temperature Trip', [83].Code := 643, [83].Desc := 'Transformer Over Temperature Warning', [84].Code := 644, [84].Desc := 'Power Cell Cabinet Fan Fault', [85].Code := 645, [85].Desc := 'Power Cell Cabinet Fan CB Open', [86].Code := 646, [86].Desc := 'Transformer Cabinet Fan Fault', [87].Code := 647, [87].Desc := 'Transformer Cabinet Fan CB Open', [88].Code := 648, [88].Desc := 'Auxiliary Power Off', [89].Code := 649, [89].Desc := 'Cabinet Door Open', [90].Code := 650,
        [90].Desc := 'External Control Power Loss Warning', [91].Code := 651, [91].Desc := 'Analog Channel #1 Loss Warning', [92].Code := 652, [92].Desc := 'DSP Communication Error', [93].Code := 653, [93].Desc := 'Cooling Fan Contactor Open', [94].Code := 559, [94].Desc := 'Versions Of System Not Compatible', [95].Code := 561, [95].Desc := 'Overtemp Time Out In Power Cell #1', [96].Code := 562, [96].Desc := 'Overtemp Time Out In Power Cell #2', [97].Code := 563, [97].Desc := 'Overtemp Time Out In Power Cell #3', [98].Code := 564, [98].Desc := 'Overtemp Time Out In Power Cell #4', [99].Code := 565, [99].Desc := 'Overtemp Time Out In Power Cell #5', [100].Code := 566, [100].Desc := 'Overtemp Time Out In Power Cell #6', [101].Code := 567, [101].Desc := 'Overtemp Time Out In Power Cell #7', [102].Code := 568, [102].Desc := 'Overtemp Time Out In Power Cell #8', [103].Code := 569, [103].Desc := 'Overtemp Time Out In Power Cell #9', [104].Code := 570, [104].Desc := 'Overtemp Time Out In Power Cell #10', [105].Code := 571, [105].Desc := 'Overtemp Time Out In Power Cell #11', [106].Code := 572, [106].Desc := 'Overtemp Time Out In Power Cell #12', [107].Code := 573, [107].Desc := 'Overtemp Time Out In Power Cell #13', [108].Code := 574, [108].Desc := 'Overtemp Time Out In Power Cell #14', [109].Code := 575, [109].Desc := 'Overtemp Time Out In Power Cell #15', [110].Code := 576, [110].Desc := 'Overtemp Time Out In Power Cell #16', [111].Code := 577, [111].Desc := 'Overtemp Time Out In Power Cell #17', [112].Code := 578, [112].Desc := 'Overtemp Time Out In Power Cell #18', [113].Code := 579, [113].Desc := 'Overtemp Time Out In Power Cell #19', [114].Code := 580, [114].Desc := 'Overtemp Time Out In Power Cell #20', [115].Code := 581, [115].Desc := 'Overtemp Time Out In Power Cell #21', [116].Code := 582, [116].Desc := 'Overtemp Time Out In Power Cell #22', [117].Code := 583, [117].Desc := 'Overtemp Time Out In Power Cell #23', [118].Code := 584, [118].Desc := 'Overtemp Time Out In Power Cell #24', [119].Code := 585, [119].Desc := 'Overtemp Time Out In Power Cell #25', [120].Code := 586,
        [120].Desc := 'Overtemp Time Out In Power Cell #26', [121].Code := 587, [121].Desc := 'Overtemp Time Out In Power Cell #27', [122].Code := 1, [122].Desc := 'IGBT Over Current In Power Cell #1', [123].Code := 2, [123].Desc := 'Capacitor Abnormal In Power Cell #1', [124].Code := 3, [124].Desc := 'Input Over Voltage In Power Cell #1', [125].Code := 4, [125].Desc := 'DC Bus Undervoltage In Power Cell #1', [126].Code := 5, [126].Desc := 'Communication Error In Power Cell #1', [127].Code := 6, [127].Desc := 'No PWM Pulse For IGBT In Power Cell #1', [128].Code := 7, [128].Desc := 'Bypass Hardware Fault In Power Cell #1', [129].Code := 8, [129].Desc := 'Comm Link Fault In Power Cell #1', [130].Code := 9, [130].Desc := 'PCCB Ver. Inompatible In Power Cell #1', [131].Code := 10, [131].Desc := 'Power Cell #1 Bypassed', [132].Code := 11, [132].Desc := 'Over Temperature In Power Cell #1', [133].Code := 12, [133].Desc := 'Power Cell #1 Failed To Bypass', [134].Code := 13, [134].Desc := 'One Phase Lost In Power Cell #1', [135].Code := 14, [135].Desc := 'Two Phases Lost In Power Cell #1', [136].Code := 15, [136].Desc := 'Bypass Failure (OV) In Power Cell #1', [137].Code := 17, [137].Desc := 'IGBT Over Current In Power Cell #2', [138].Code := 18, [138].Desc := 'Capacitor Abnormal In Power Cell #2', [139].Code := 19, [139].Desc := 'Input Over Voltage In Power Cell #2', [140].Code := 20, [140].Desc := 'DC Bus Undervoltage In Power Cell #2', [141].Code := 21, [141].Desc := 'Communication Error In Power Cell #2', [142].Code := 22, [142].Desc := 'No PWM Pulse For IGBT In Power Cell #2', [143].Code := 23, [143].Desc := 'Bypass Hardware Fault In Power Cell #2', [144].Code := 24, [144].Desc := 'Comm Link Fault in Power Cell #2', [145].Code := 25, [145].Desc := 'PCCB Ver. Incompatible In Power Cell #2', [146].Code := 26, [146].Desc := 'Power Cell #2 Bypassed', [147].Code := 27, [147].Desc := 'Over Temperature In Power Cell #2', [148].Code := 28, [148].Desc := 'Power Cell #2 Failed To Bypass', [149].Code := 29, [149].Desc := 'One Phase Lost In Power Cell #2', [150].Code := 30,
        [150].Desc := 'Two Phases Lost In Power Cell #2', [151].Code := 31, [151].Desc := 'Bypass Failure (OV) In Power Cell #2', [152].Code := 33, [152].Desc := 'IGBT Over Current In Power Cell #3', [153].Code := 34, [153].Desc := 'Capacitor Abnormal In Power Cell #3', [154].Code := 35, [154].Desc := 'Input Over Voltage In Power Cell #3', [155].Code := 36, [155].Desc := 'DC Bus Undervoltage In Power Cell #3', [156].Code := 37, [156].Desc := 'Communication Error In Power Cell #3', [157].Code := 38, [157].Desc := 'No PWM Pulse For IGBT In Power Cell #3', [158].Code := 39, [158].Desc := 'Bypass Hardware Fault In Power Cell #3', [159].Code := 40, [159].Desc := 'Comm Link Fault in Power Cell #3', [160].Code := 41, [160].Desc := 'PCCB Ver. Incompatible In Power Cell #3', [161].Code := 42, [161].Desc := 'Power Cell #3 Bypassed', [162].Code := 43, [162].Desc := 'Over Temperature In Power Cell #3', [163].Code := 44, [163].Desc := 'Power Cell #3 Failed To Bypass', [164].Code := 45, [164].Desc := 'One Phase Lost In Power Cell #3', [165].Code := 46, [165].Desc := 'Two Phases Lost In Power Cell #3', [166].Code := 47, [166].Desc := 'Bypass Failure (OV) In Power Cell #3', [167].Code := 49, [167].Desc := 'IGBT Over Current In Power Cell #4', [168].Code := 50, [168].Desc := 'Capacitor Abnormal In Power Cell #4', [169].Code := 51, [169].Desc := 'Input Over Voltage In Power Cell #4', [170].Code := 52, [170].Desc := 'DC Bus Undervoltage In Power Cell #4', [171].Code := 53, [171].Desc := 'Communication Error In Power Cell #4', [172].Code := 54, [172].Desc := 'No PWM Pulse For IGBT In Power Cell #4', [173].Code := 55, [173].Desc := 'Bypass Hardware Fault In Power Cell #4', [174].Code := 56, [174].Desc := 'Comm Link Fault in Power Cell #4', [175].Code := 57, [175].Desc := 'PCCB Ver. Incompatible In Power Cell #4', [176].Code := 58, [176].Desc := 'Power Cell #4 Bypassed', [177].Code := 59, [177].Desc := 'Over Temperature In Power Cell #4', [178].Code := 60, [178].Desc := 'Power Cell #4 Failed To Bypass', [179].Code := 61, [179].Desc := 'One Phase Lost In Power Cell #4', [180].Code := 62,
        [180].Desc := 'Two Phases Lost In Power Cell #4', [181].Code := 63, [181].Desc := 'Bypass Failure (OV) In Power Cell #4', [182].Code := 65, [182].Desc := 'IGBT Over Current In Power Cell #5', [183].Code := 66, [183].Desc := 'Capacitor Abnormal In Power Cell #5', [184].Code := 67, [184].Desc := 'Input Over Voltage In Power Cell #5', [185].Code := 68, [185].Desc := 'DC Bus Undervoltage In Power Cell #5', [186].Code := 69, [186].Desc := 'Communication Error In Power Cell #5', [187].Code := 70, [187].Desc := 'No PWM Pulse For IGBT In Power Cell #5', [188].Code := 71, [188].Desc := 'Bypass Hardware Fault In Power Cell #5', [189].Code := 72, [189].Desc := 'Comm Link Fault in Power Cell #5', [190].Code := 73, [190].Desc := 'PCCB Ver. Incompatible In Power Cell #5', [191].Code := 74, [191].Desc := 'Power Cell #5 Bypassed', [192].Code := 75, [192].Desc := 'Over Temperature In Power Cell #5', [193].Code := 76, [193].Desc := 'Power Cell #5 Failed To Bypass', [194].Code := 77, [194].Desc := 'One Phase Lost In Power Cell #5', [195].Code := 78, [195].Desc := 'Two Phases Lost In Power Cell #5', [196].Code := 79, [196].Desc := 'Bypass Failure (OV) In Power Cell #5', [197].Code := 81, [197].Desc := 'IGBT Over Current In Power Cell #6', [198].Code := 82, [198].Desc := 'Capacitor Abnormal In Power Cell #6', [199].Code := 83, [199].Desc := 'Input Over Voltage In Power Cell #6', [200].Code := 84, [200].Desc := 'DC Bus Undervoltage In Power Cell #6', [201].Code := 85, [201].Desc := 'Communication Error In Power Cell #6', [202].Code := 86, [202].Desc := 'No PWM Pulse For IGBT In Power Cell #6', [203].Code := 87, [203].Desc := 'Bypass Hardware Fault In Power Cell #6', [204].Code := 88, [204].Desc := 'Comm Link Fault in Power Cell #6', [205].Code := 89, [205].Desc := 'PCCB Ver. Incompatible In Power Cell #6', [206].Code := 90, [206].Desc := 'Power Cell #6 Bypassed', [207].Code := 91, [207].Desc := 'Over Temperature In Power Cell #6', [208].Code := 92, [208].Desc := 'Power Cell #6 Failed To Bypass', [209].Code := 93, [209].Desc := 'One Phase Lost In Power Cell #6', [210].Code := 94,
        [210].Desc := 'Two Phases Lost In Power Cell #6', [211].Code := 95, [211].Desc := 'Bypass Failure (OV) In Power Cell #6', [212].Code := 97, [212].Desc := 'IGBT Over Current In Power Cell #7', [213].Code := 98, [213].Desc := 'Capacitor Abnormal In Power Cell #7', [214].Code := 99, [214].Desc := 'Input Over Voltage In Power Cell #7', [215].Code := 100, [215].Desc := 'DC Bus Undervoltage In Power Cell #7', [216].Code := 101, [216].Desc := 'Communication Error In Power Cell #7', [217].Code := 102, [217].Desc := 'No PWM Pulse For IGBT In Power Cell #7', [218].Code := 103, [218].Desc := 'Bypass Hardware Fault In Power Cell #7', [219].Code := 104, [219].Desc := 'Comm Link Fault in Power Cell #7', [220].Code := 105, [220].Desc := 'PCCB Ver. Incompatible In Power Cell #7', [221].Code := 106, [221].Desc := 'Power Cell #7 Bypassed', [222].Code := 107, [222].Desc := 'Over Temperature In Power Cell #7', [223].Code := 108, [223].Desc := 'Power Cell #7 Failed To Bypass', [224].Code := 109, [224].Desc := 'One Phase Lost In Power Cell #7', [225].Code := 110, [225].Desc := 'Two Phases Lost In Power Cell #7', [226].Code := 111, [226].Desc := 'Bypass Failure (OV) In Power Cell #7', [227].Code := 113, [227].Desc := 'IGBT Over Current In Power Cell #8', [228].Code := 114, [228].Desc := 'Capacitor Abnormal In Power Cell #8', [229].Code := 115, [229].Desc := 'Input Over Voltage In Power Cell #8', [230].Code := 116, [230].Desc := 'DC Bus Undervoltage In Power Cell #8', [231].Code := 117, [231].Desc := 'Communication Error In Power Cell #8', [232].Code := 118, [232].Desc := 'No PWM Pulse For IGBT In Power Cell #8', [233].Code := 119, [233].Desc := 'Bypass Hardware Fault In Power Cell #8', [234].Code := 120, [234].Desc := 'Comm Link Fault in Power Cell #8', [235].Code := 121, [235].Desc := 'PCCB Ver. Incompatible In Power Cell #8', [236].Code := 122, [236].Desc := 'Power Cell #8 Bypassed', [237].Code := 123, [237].Desc := 'Over Temperature In Power Cell #8', [238].Code := 124, [238].Desc := 'Power Cell #8 Failed To Bypass', [239].Code := 125, [239].Desc := 'One Phase Lost In Power Cell #8', [240].Code := 126,
        [240].Desc := 'Two Phases Lost In Power Cell #8', [241].Code := 127, [241].Desc := 'Bypass Failure (OV) In Power Cell #8', [242].Code := 129, [242].Desc := 'IGBT Over Current In Power Cell #9', [243].Code := 130, [243].Desc := 'Capacitor Abnormal In Power Cell #9', [244].Code := 131, [244].Desc := 'Input Over Voltage In Power Cell #9', [245].Code := 132, [245].Desc := 'DC Bus Undervoltage In Power Cell #9', [246].Code := 133, [246].Desc := 'Communication Error In Power Cell #9', [247].Code := 134, [247].Desc := 'No PWM Pulse For IGBT In Power Cell #9', [248].Code := 135, [248].Desc := 'Bypass Hardware Fault In Power Cell #9', [249].Code := 136, [249].Desc := 'Comm Link Fault in Power Cell #9', [250].Code := 137, [250].Desc := 'PCCB Ver. Incompatible In Power Cell #9', [251].Code := 138, [251].Desc := 'Power Cell #9 Bypassed', [252].Code := 139, [252].Desc := 'Over Temperature In Power Cell #9', [253].Code := 140, [253].Desc := 'Power Cell #9 Failed To Bypass', [254].Code := 141, [254].Desc := 'One Phase Lost In Power Cell #9', [255].Code := 142, [255].Desc := 'Two Phases Lost In Power Cell #9', [256].Code := 143, [256].Desc := 'Bypass Failure (OV) In Power Cell #9', [257].Code := 145, [257].Desc := 'IGBT Over Current In Power Cell #10', [258].Code := 146, [258].Desc := 'Capacitor Abnormal In Power Cell #10', [259].Code := 147, [259].Desc := 'Input Over Voltage In Power Cell #10', [260].Code := 148, [260].Desc := 'DC Bus Undervoltage In Power Cell #10', [261].Code := 149, [261].Desc := 'Communication Error In Power Cell #10', [262].Code := 150, [262].Desc := 'No PWM Pulse For IGBT In Power Cell #10', [263].Code := 151, [263].Desc := 'Bypass Hardware Fault In Power Cell #10', [264].Code := 152, [264].Desc := 'Comm Link Fault in Power Cell #10', [265].Code := 153, [265].Desc := 'PCCB Ver. Incompatible In Power Cell #10', [266].Code := 154, [266].Desc := 'Power Cell #10 Bypassed', [267].Code := 155, [267].Desc := 'Over Temperature In Power Cell #10', [268].Code := 156, [268].Desc := 'Power Cell #10 Failed To Bypass', [269].Code := 157, [269].Desc := 'One Phase Lost In Power Cell #10', [270].Code := 158,
        [270].Desc := 'Two Phases Lost In Power Cell #10', [271].Code := 159, [271].Desc := 'Bypass Failure (OV) In Power Cell #10', [272].Code := 161, [272].Desc := 'IGBT Over Current In Power Cell #11', [273].Code := 162, [273].Desc := 'Capacitor Abnormal In Power Cell #11', [274].Code := 163, [274].Desc := 'Input Over Voltage In Power Cell #11', [275].Code := 164, [275].Desc := 'DC Bus Undervoltage In Power Cell #11', [276].Code := 165, [276].Desc := 'Communication Error In Power Cell #11', [277].Code := 166, [277].Desc := 'No PWM Pulse For IGBT In Power Cell #11', [278].Code := 167, [278].Desc := 'Bypass Hardware Fault In Power Cell #11', [279].Code := 168, [279].Desc := 'Comm Link Fault in Power Cell #11', [280].Code := 169, [280].Desc := 'PCCB Ver. Incompatible In Power Cell #11', [281].Code := 170, [281].Desc := 'Power Cell #11 Bypassed', [282].Code := 171, [282].Desc := 'Over Temperature In Power Cell #11', [283].Code := 172, [283].Desc := 'Power Cell #11 Failed To Bypass', [284].Code := 173, [284].Desc := 'One Phase Lost In Power Cell #11', [285].Code := 174, [285].Desc := 'Two Phases Lost In Power Cell #11', [286].Code := 175, [286].Desc := 'Bypass Failure (OV) In Power Cell #11', [287].Code := 177, [287].Desc := 'IGBT Over Current In Power Cell #12', [288].Code := 178, [288].Desc := 'Capacitor Abnormal In Power Cell #12', [289].Code := 179, [289].Desc := 'Input Over Voltage In Power Cell #12', [290].Code := 180, [290].Desc := 'DC Bus Undervoltage In Power Cell #12', [291].Code := 181, [291].Desc := 'Communication Error In Power Cell #12', [292].Code := 182, [292].Desc := 'No PWM Pulse For IGBT In Power Cell #12', [293].Code := 183, [293].Desc := 'Bypass Hardware Fault In Power Cell #12', [294].Code := 184, [294].Desc := 'Comm Link Fault in Power Cell #12', [295].Code := 185, [295].Desc := 'PCCB Ver. Incompatible In Power Cell #12', [296].Code := 186, [296].Desc := 'Power Cell #12 Bypassed', [297].Code := 187, [297].Desc := 'Over Temperature In Power Cell #12', [298].Code := 188, [298].Desc := 'Power Cell #12 Failed To Bypass', [299].Code := 189, [299].Desc := 'One Phase Lost In Power Cell #12', [300].Code := 190,
        [300].Desc := 'Two Phases Lost In Power Cell #12', [301].Code := 191, [301].Desc := 'Bypass Failure (OV) In Power Cell #12', [302].Code := 193, [302].Desc := 'IGBT Over Current In Power Cell #13', [303].Code := 194, [303].Desc := 'Capacitor Abnormal In Power Cell #13', [304].Code := 195, [304].Desc := 'Input Over Voltage In Power Cell #13', [305].Code := 196, [305].Desc := 'DC Bus Undervoltage In Power Cell #13', [306].Code := 197, [306].Desc := 'Communication Error In Power Cell #13', [307].Code := 198, [307].Desc := 'No PWM Pulse For IGBT In Power Cell #13', [308].Code := 199, [308].Desc := 'Bypass Hardware Fault In Power Cell #13', [309].Code := 200, [309].Desc := 'Comm Link Fault in Power Cell #13', [310].Code := 201, [310].Desc := 'PCCB Ver. Incompatible In Power Cell #13', [311].Code := 202, [311].Desc := 'Power Cell #13 Bypassed', [312].Code := 203, [312].Desc := 'Over Temperature In Power Cell #13', [313].Code := 204, [313].Desc := 'Power Cell #13 Failed To Bypass', [314].Code := 205, [314].Desc := 'One Phase Lost In Power Cell #13', [315].Code := 206, [315].Desc := 'Two Phases Lost In Power Cell #13', [316].Code := 207, [316].Desc := 'Bypass Failure (OV) In Power Cell #13', [317].Code := 209, [317].Desc := 'IGBT Over Current In Power Cell #14', [318].Code := 210, [318].Desc := 'Capacitor Abnormal In Power Cell #14', [319].Code := 211, [319].Desc := 'Input Over Voltage In Power Cell #14', [320].Code := 212, [320].Desc := 'DC Bus Undervoltage In Power Cell #14', [321].Code := 213, [321].Desc := 'Communication Error In Power Cell #14', [322].Code := 214, [322].Desc := 'No PWM Pulse For IGBT In Power Cell #14', [323].Code := 215, [323].Desc := 'Bypass Hardware Fault In Power Cell #14', [324].Code := 216, [324].Desc := 'Comm Link Fault in Power Cell #14', [325].Code := 217, [325].Desc := 'PCCB Ver. Incompatible In Power Cell #14', [326].Code := 218, [326].Desc := 'Power Cell #14 Bypassed', [327].Code := 219, [327].Desc := 'Over Temperature In Power Cell #14', [328].Code := 220, [328].Desc := 'Power Cell #14 Failed To Bypass', [329].Code := 221, [329].Desc := 'One Phase Lost In Power Cell #14', [330].Code := 222,
        [330].Desc := 'Two Phases Lost In Power Cell #14', [331].Code := 223, [331].Desc := 'Bypass Failure (OV) In Power Cell #14', [332].Code := 225, [332].Desc := 'IGBT Over Current In Power Cell #15', [333].Code := 226, [333].Desc := 'Capacitor Abnormal In Power Cell #15', [334].Code := 227, [334].Desc := 'Input Over Voltage In Power Cell #15', [335].Code := 228, [335].Desc := 'DC Bus Undervoltage In Power Cell #15', [336].Code := 229, [336].Desc := 'Communication Error In Power Cell #15', [337].Code := 230, [337].Desc := 'No PWM Pulse For IGBT In Power Cell #15', [338].Code := 231, [338].Desc := 'Bypass Hardware Fault In Power Cell #15', [339].Code := 232, [339].Desc := 'Comm Link Fault in Power Cell #15', [340].Code := 233, [340].Desc := 'PCCB Ver. Incompatible In Power Cell #15', [341].Code := 234, [341].Desc := 'Power Cell #15 Bypassed', [342].Code := 235, [342].Desc := 'Over Temperature In Power Cell #15', [343].Code := 236, [343].Desc := 'Power Cell #15 Failed To Bypass', [344].Code := 237, [344].Desc := 'One Phase Lost In Power Cell #15', [345].Code := 238, [345].Desc := 'Two Phases Lost In Power Cell #15', [346].Code := 239, [346].Desc := 'Bypass Failure (OV) In Power Cell #15', [347].Code := 241, [347].Desc := 'IGBT Over Current In Power Cell #16', [348].Code := 242, [348].Desc := 'Capacitor Abnormal In Power Cell #16', [349].Code := 243, [349].Desc := 'Input Over Voltage In Power Cell #16', [350].Code := 244, [350].Desc := 'DC Bus Undervoltage In Power Cell #16', [351].Code := 245, [351].Desc := 'Communication Error In Power Cell #16', [352].Code := 246, [352].Desc := 'No PWM Pulse For IGBT In Power Cell #16', [353].Code := 247, [353].Desc := 'Bypass Hardware Fault In Power Cell #16', [354].Code := 248, [354].Desc := 'Comm Link Fault in Power Cell #16', [355].Code := 249, [355].Desc := 'PCCB Ver. Incompatible In Power Cell #16', [356].Code := 250, [356].Desc := 'Power Cell #16 Bypassed', [357].Code := 251, [357].Desc := 'Over Temperature In Power Cell #16', [358].Code := 252, [358].Desc := 'Power Cell #16 Failed To Bypass', [359].Code := 253, [359].Desc := 'One Phase Lost In Power Cell #16', [360].Code := 254,
        [360].Desc := 'Two Phases Lost In Power Cell #16', [361].Code := 255, [361].Desc := 'Bypass Failure (OV) In Power Cell #16', [362].Code := 257, [362].Desc := 'IGBT Over Current In Power Cell #17', [363].Code := 258, [363].Desc := 'Capacitor Abnormal In Power Cell #17', [364].Code := 259, [364].Desc := 'Input Over Voltage In Power Cell #17', [365].Code := 260, [365].Desc := 'DC Bus Undervoltage In Power Cell #17', [366].Code := 261, [366].Desc := 'Communication Error In Power Cell #17', [367].Code := 262, [367].Desc := 'No PWM Pulse For IGBT In Power Cell #17', [368].Code := 263, [368].Desc := 'Bypass Hardware Fault In Power Cell #17', [369].Code := 264, [369].Desc := 'Comm Link Fault in Power Cell #17', [370].Code := 265, [370].Desc := 'PCCB Ver. Incompatible In Power Cell #17', [371].Code := 266, [371].Desc := 'Power Cell #17 Bypassed', [372].Code := 267, [372].Desc := 'Over Temperature In Power Cell #17', [373].Code := 268, [373].Desc := 'Power Cell #17 Failed To Bypass', [374].Code := 269, [374].Desc := 'One Phase Lost In Power Cell #17', [375].Code := 270, [375].Desc := 'Two Phases Lost In Power Cell #17', [376].Code := 271, [376].Desc := 'Bypass Failure (OV) In Power Cell #17', [377].Code := 273, [377].Desc := 'IGBT Over Current In Power Cell #18', [378].Code := 274, [378].Desc := 'Capacitor Abnormal In Power Cell #18', [379].Code := 275, [379].Desc := 'Input Over Voltage In Power Cell #18', [380].Code := 276, [380].Desc := 'DC Bus Undervoltage In Power Cell #18', [381].Code := 277, [381].Desc := 'Communication Error In Power Cell #18', [382].Code := 278, [382].Desc := 'No PWM Pulse For IGBT In Power Cell #18', [383].Code := 279, [383].Desc := 'Bypass Hardware Fault In Power Cell #18', [384].Code := 280, [384].Desc := 'Comm Link Fault in Power Cell #18', [385].Code := 281, [385].Desc := 'PCCB Ver. Incompatible In Power Cell #18', [386].Code := 282, [386].Desc := 'Power Cell #18 Bypassed', [387].Code := 283, [387].Desc := 'Over Temperature In Power Cell #18', [388].Code := 284, [388].Desc := 'Power Cell #18 Failed To Bypass', [389].Code := 285, [389].Desc := 'One Phase Lost In Power Cell #18', [390].Code := 286,
        [390].Desc := 'Two Phases Lost In Power Cell #18', [391].Code := 287, [391].Desc := 'Bypass Failure (OV) In Power Cell #18', [392].Code := 289, [392].Desc := 'IGBT Over Current In Power Cell #19', [393].Code := 290, [393].Desc := 'Capacitor Abnormal In Power Cell #19', [394].Code := 291, [394].Desc := 'Input Over Voltage In Power Cell #19', [395].Code := 292, [395].Desc := 'DC Bus Undervoltage In Power Cell #19', [396].Code := 293, [396].Desc := 'Communication Error In Power Cell #19', [397].Code := 294, [397].Desc := 'No PWM Pulse For IGBT In Power Cell #19', [398].Code := 295, [398].Desc := 'Bypass Hardware Fault In Power Cell #19', [399].Code := 296, [399].Desc := 'Comm Link Fault in Power Cell #19', [400].Code := 297, [400].Desc := 'PCCB Ver. Incompatible In Power Cell #19', [401].Code := 298, [401].Desc := 'Power Cell #19 Bypassed', [402].Code := 299, [402].Desc := 'Over Temperature In Power Cell #19', [403].Code := 300, [403].Desc := 'Power Cell #19 Failed To Bypass', [404].Code := 301, [404].Desc := 'One Phase Lost In Power Cell #19', [405].Code := 302, [405].Desc := 'Two Phases Lost In Power Cell #19', [406].Code := 303, [406].Desc := 'Bypass Failure (OV) In Power Cell #19', [407].Code := 305, [407].Desc := 'IGBT Over Current In Power Cell #20', [408].Code := 306, [408].Desc := 'Capacitor Abnormal In Power Cell #20', [409].Code := 307, [409].Desc := 'Input Over Voltage In Power Cell #20', [410].Code := 308, [410].Desc := 'DC Bus Undervoltage In Power Cell #20', [411].Code := 309, [411].Desc := 'Communication Error In Power Cell #20', [412].Code := 310, [412].Desc := 'No PWM Pulse For IGBT In Power Cell #20', [413].Code := 311, [413].Desc := 'Bypass Hardware Fault In Power Cell #20', [414].Code := 312, [414].Desc := 'Comm Link Fault in Power Cell #20', [415].Code := 313, [415].Desc := 'PCCB Ver. Incompatible In Power Cell #20', [416].Code := 314, [416].Desc := 'Power Cell #20 Bypassed', [417].Code := 315, [417].Desc := 'Over Temperature In Power Cell #20', [418].Code := 316, [418].Desc := 'Power Cell #20 Failed To Bypass', [419].Code := 317, [419].Desc := 'One Phase Lost In Power Cell #20', [420].Code := 318,
        [420].Desc := 'Two Phases Lost In Power Cell #20', [421].Code := 319, [421].Desc := 'Bypass Failure (OV) In Power Cell #20', [422].Code := 321, [422].Desc := 'IGBT Over Current In Power Cell #21', [423].Code := 322, [423].Desc := 'Capacitor Abnormal In Power Cell #21', [424].Code := 323, [424].Desc := 'Input Over Voltage In Power Cell #21', [425].Code := 324, [425].Desc := 'DC Bus Undervoltage In Power Cell #21', [426].Code := 325, [426].Desc := 'Communication Error In Power Cell #21', [427].Code := 326, [427].Desc := 'No PWM Pulse For IGBT In Power Cell #21', [428].Code := 327, [428].Desc := 'Bypass Hardware Fault In Power Cell #21', [429].Code := 328, [429].Desc := 'Comm Link Fault in Power Cell #21', [430].Code := 329, [430].Desc := 'PCCB Ver. Incompatible In Power Cell #21', [431].Code := 330, [431].Desc := 'Power Cell #21 Bypassed', [432].Code := 331, [432].Desc := 'Over Temperature In Power Cell #21', [433].Code := 332, [433].Desc := 'Power Cell #21 Failed To Bypass', [434].Code := 333, [434].Desc := 'One Phase Lost In Power Cell #21', [435].Code := 334, [435].Desc := 'Two Phases Lost In Power Cell #21', [436].Code := 335, [436].Desc := 'Bypass Failure (OV) In Power Cell #21', [437].Code := 337, [437].Desc := 'IGBT Over Current In Power Cell #22', [438].Code := 338, [438].Desc := 'Capacitor Abnormal In Power Cell #22', [439].Code := 339, [439].Desc := 'Input Over Voltage In Power Cell #22', [440].Code := 340, [440].Desc := 'DC Bus Undervoltage In Power Cell #22', [441].Code := 341, [441].Desc := 'Communication Error In Power Cell #22', [442].Code := 342, [442].Desc := 'No PWM Pulse For IGBT In Power Cell #22', [443].Code := 343, [443].Desc := 'Bypass Hardware Fault In Power Cell #22', [444].Code := 344, [444].Desc := 'Comm Link Fault in Power Cell #22', [445].Code := 345, [445].Desc := 'PCCB Ver. Incompatible In Power Cell #22', [446].Code := 346, [446].Desc := 'Power Cell #22 Bypassed', [447].Code := 347, [447].Desc := 'Over Temperature In Power Cell #22', [448].Code := 348, [448].Desc := 'Power Cell #22 Failed To Bypass', [449].Code := 349, [449].Desc := 'One Phase Lost In Power Cell #22', [450].Code := 350,
